LIN {X 0.099,Y -360.275,Z 1680.409,A 0.000,B 0.000,C 90.000,E1 73.630} C_DIS
LIN {X 0.182,Y -346.162,Z 1680.394,A 0.000,B 0.000,C 90.000,E1 70.913} C_DIS
LIN {X 0.106,Y -331.569,Z 1680.377,A 0.000,B 0.000,C 90.000,E1 67.847} C_DIS
LIN {X -0.099,Y -319.051,Z 1680.361,A 0.000,B 0.000,C 90.000,E1 65.049} C_DIS
LIN {X -0.146,Y -308.197,Z 1680.347,A 0.000,B 0.000,C 90.000,E1 62.487} C_DIS
LIN {X -0.186,Y -298.755,Z 1680.334,A 0.000,B 0.000,C 90.000,E1 60.205} C_DIS
LIN {X -0.133,Y -290.521,Z 1680.323,A 0.000,B 0.000,C 90.000,E1 58.201} C_DIS
LIN {X 0.074,Y -282.040,Z 1680.312,A 0.000,B 0.000,C 90.000,E1 56.135} C_DIS
LIN {X -0.110,Y -273.413,Z 1680.301,A 0.000,B 0.000,C 90.000,E1 54.116} C_DIS
LIN {X -0.060,Y -263.348,Z 1680.287,A 0.000,B 0.000,C 90.000,E1 51.662} C_DIS
LIN {X -0.034,Y -250.950,Z 1680.269,A 0.000,B 0.000,C 90.000,E1 48.447} C_DIS
LIN {X -0.049,Y -239.332,Z 1680.251,A 0.000,B 0.000,C 90.000,E1 45.162} C_DIS
LIN {X 0.006,Y -229.929,Z 1680.234,A 0.000,B 0.000,C 90.000,E1 42.162} C_DIS
LIN {X 0.085,Y -222.365,Z 1680.219,A 0.000,B 0.000,C 90.000,E1 39.483} C_DIS
LIN {X -0.012,Y -214.434,Z 1680.202,A 0.000,B 0.000,C 90.000,E1 36.423} C_DIS
LIN {X -0.034,Y -207.223,Z 1680.185,A 0.000,B 0.000,C 90.000,E1 33.293} C_DIS
LIN {X 0.067,Y -200.567,Z 1680.167,A 0.000,B 0.000,C 90.000,E1 30.079} C_DIS
LIN {X -0.020,Y -194.422,Z 1680.149,A 0.000,B 0.000,C 90.000,E1 26.873} C_DIS
LIN {X 0.005,Y -188.845,Z 1680.131,A 0.000,B 0.000,C 90.000,E1 23.590} C_DIS
LIN {X -0.084,Y -183.863,Z 1680.113,A 0.000,B 0.000,C 90.000,E1 20.301} C_DIS
LIN {X 0.028,Y -179.445,Z 1680.094,A 0.000,B 0.000,C 90.000,E1 16.913} C_DIS
LIN {X -0.003,Y -175.792,Z 1680.075,A 0.000,B 0.000,C 90.000,E1 13.536} C_DIS
LIN {X -0.006,Y -172.211,Z 1680.052,A 0.000,B 0.000,C 90.000,E1 9.265} C_DIS
LIN {X 0.053,Y -169.093,Z 1680.023,A 0.000,B 0.000,C 90.000,E1 4.073} C_DIS
LIN {X 0.081,Y -167.205,Z 1679.988,A 0.000,B 0.000,C 90.000,E1 357.764} C_DIS
LIN {X -0.016,Y -168.352,Z 1679.930,A 0.000,B 0.000,C 90.000,E1 347.353} C_DIS
LIN {X 0.061,Y -170.991,Z 1679.901,A 0.000,B 0.000,C 90.000,E1 342.127} C_DIS
LIN {X -0.022,Y -174.386,Z 1679.877,A 0.000,B 0.000,C 90.000,E1 337.847} C_DIS
LIN {X 0.038,Y -178.074,Z 1679.858,A 0.000,B 0.000,C 90.000,E1 334.409} C_DIS
LIN {X -0.065,Y -182.436,Z 1679.839,A 0.000,B 0.000,C 90.000,E1 331.051} C_DIS
LIN {X 0.050,Y -187.733,Z 1679.820,A 0.000,B 0.000,C 90.000,E1 327.661} C_DIS
LIN {X 0.015,Y -192.363,Z 1679.807,A 0.000,B 0.000,C 90.000,E1 325.182} C_DIS
LIN {X 0.016,Y -197.628,Z 1679.793,A 0.000,B 0.000,C 90.000,E1 322.718} C_DIS
LIN {X -0.080,Y -204.609,Z 1679.777,A 0.000,B 0.000,C 90.000,E1 319.908} C_DIS
LIN {X -0.032,Y -212.531,Z 1679.762,A 0.000,B 0.000,C 90.000,E1 317.106} C_DIS
LIN {X 0.028,Y -221.548,Z 1679.746,A 0.000,B 0.000,C 90.000,E1 314.352} C_DIS
LIN {X -0.018,Y -231.549,Z 1679.732,A 0.000,B 0.000,C 90.000,E1 311.676} C_DIS
LIN {X 0.050,Y -241.118,Z 1679.719,A 0.000,B 0.000,C 90.000,E1 309.402} C_DIS
LIN {X -0.006,Y -251.816,Z 1679.707,A 0.000,B 0.000,C 90.000,E1 307.202} C_DIS
LIN {X -0.009,Y -267.871,Z 1679.691,A 0.000,B 0.000,C 90.000,E1 304.326} C_DIS
LIN {X 0.014,Y -283.371,Z 1679.677,A 0.000,B 0.000,C 90.000,E1 301.878} C_DIS
LIN {X -0.162,Y -300.081,Z 1679.664,A 0.000,B 0.000,C 90.000,E1 299.539} C_DIS
LIN {X 0.012,Y -317.510,Z 1679.651,A 0.000,B 0.000,C 90.000,E1 297.206} C_DIS
LIN {X 0.091,Y -330.014,Z 1679.642,A 0.000,B 0.000,C 90.000,E1 295.591} C_DIS
LIN {X -0.088,Y -347.481,Z 1679.630,A 0.000,B 0.000,C 90.000,E1 293.439} C_DIS
LIN {X 0.040,Y -360.043,Z 1679.622,A 0.000,B 0.000,C 90.000,E1 291.897} C_DIS
LIN {X -0.092,Y -372.166,Z 1679.613,A 0.000,B 0.000,C 90.000,E1 290.429} C_DIS
LIN {X 0.075,Y -378.963,Z 1679.609,A 0.000,B 0.000,C 90.000,E1 289.523} C_DIS
LIN {X -0.042,Y -385.176,Z 1679.604,A 0.000,B 0.000,C 90.000,E1 288.671} C_DIS
LIN {X -0.115,Y -390.636,Z 1679.599,A 0.000,B 0.000,C 90.000,E1 287.819} C_DIS
LIN {X -0.137,Y -395.273,Z 1679.594,A 0.000,B 0.000,C 90.000,E1 286.968} C_DIS
LIN {X 0.145,Y -398.887,Z 1679.589,A 0.000,B 0.000,C 90.000,E1 286.079} C_DIS
LIN {X -0.099,Y -400.856,Z 1679.586,A 0.000,B 0.000,C 90.000,E1 285.552} C_DIS
LIN {X 0.157,Y -402.461,Z 1679.583,A 0.000,B 0.000,C 90.000,E1 284.954} C_DIS
LIN {X 0.034,Y -403.719,Z 1679.580,A 0.000,B 0.000,C 90.000,E1 284.411} C_DIS
LIN {X -0.182,Y -404.584,Z 1679.577,A 0.000,B 0.000,C 90.000,E1 283.883} C_DIS
LIN {X 0.006,Y -404.997,Z 1679.574,A 0.000,B 0.000,C 90.000,E1 283.300} C_DIS
LIN {X -0.195,Y -405.069,Z 1679.571,A 0.000,B 0.000,C 90.000,E1 282.771} C_DIS
LIN {X 0.004,Y -404.620,Z 1679.568,A 0.000,B 0.000,C 90.000,E1 282.187} C_DIS
LIN {X -0.192,Y -403.716,Z 1679.565,A 0.000,B 0.000,C 90.000,E1 281.658} C_DIS
LIN {X 0.004,Y -402.255,Z 1679.562,A 0.000,B 0.000,C 90.000,E1 281.074} C_DIS
LIN {X -0.200,Y -400.281,Z 1679.558,A 0.000,B 0.000,C 90.000,E1 280.546} C_DIS
LIN {X -0.021,Y -397.689,Z 1679.555,A 0.000,B 0.000,C 90.000,E1 279.962} C_DIS
LIN {X 0.135,Y -394.640,Z 1679.552,A 0.000,B 0.000,C 90.000,E1 279.378} C_DIS
LIN {X -0.119,Y -389.406,Z 1679.547,A 0.000,B 0.000,C 90.000,E1 278.568} C_DIS
LIN {X -0.025,Y -383.414,Z 1679.543,A 0.000,B 0.000,C 90.000,E1 277.701} C_DIS
LIN {X -0.008,Y -378.966,Z 1679.540,A 0.000,B 0.000,C 90.000,E1 277.125} C_DIS
LIN {X -0.016,Y -373.970,Z 1679.536,A 0.000,B 0.000,C 90.000,E1 276.549} C_DIS
LIN {X 0.069,Y -368.403,Z 1679.533,A 0.000,B 0.000,C 90.000,E1 275.967} C_DIS
LIN {X -0.036,Y -362.598,Z 1679.530,A 0.000,B 0.000,C 90.000,E1 275.454} C_DIS
LIN {X 0.114,Y -356.440,Z 1679.527,A 0.000,B 0.000,C 90.000,E1 274.935} C_DIS
LIN {X -0.154,Y -350.104,Z 1679.525,A 0.000,B 0.000,C 90.000,E1 274.531} C_DIS
LIN {X 0.146,Y -343.492,Z 1679.523,A 0.000,B 0.000,C 90.000,E1 274.073} C_DIS
LIN {X 0.093,Y -333.687,Z 1679.520,A 0.000,B 0.000,C 90.000,E1 273.555} C_DIS
LIN {X 0.060,Y -323.811,Z 1679.517,A 0.000,B 0.000,C 90.000,E1 273.094} C_DIS
LIN {X -0.012,Y -313.990,Z 1679.515,A 0.000,B 0.000,C 90.000,E1 272.694} C_DIS
LIN {X 0.146,Y -303.822,Z 1679.513,A 0.000,B 0.000,C 90.000,E1 272.293} C_DIS
LIN {X 0.009,Y -293.379,Z 1679.511,A 0.000,B 0.000,C 90.000,E1 272.007} C_DIS
LIN {X -0.132,Y -281.634,Z 1679.510,A 0.000,B 0.000,C 90.000,E1 271.776} C_DIS
LIN {X 0.036,Y -273.036,Z 1679.509,A 0.000,B 0.000,C 90.000,E1 271.604} C_DIS
LIN {X -0.021,Y -259.535,Z 1679.508,A 0.000,B 0.000,C 90.000,E1 271.489} C_DIS
LIN {X -0.031,Y -205.689,Z 1679.508,A 0.000,B 0.000,C 90.000,E1 271.375} C_DIS
LIN {X 0.019,Y -183.367,Z 1679.507,A 0.000,B 0.000,C 90.000,E1 271.260} C_DIS
LIN {X -0.015,Y -181.401,Z 1679.507,A 0.000,B 0.000,C 90.000,E1 271.260} C_DIS
LIN {X 0.026,Y -181.581,Z 1679.501,A 0.000,B 0.000,C 90.000,E1 270.229} C_DIS
LIN {X 0.030,Y -180.865,Z 1679.472,A 0.000,B 0.000,C 90.000,E1 265.008} C_DIS
LIN {X -0.094,Y -178.980,Z 1679.444,A 0.000,B 0.000,C 90.000,E1 259.982} C_DIS
LIN {X -0.082,Y -177.950,Z 1679.435,A 0.000,B 0.000,C 90.000,E1 258.285} C_DIS
LIN {X -0.062,Y -175.591,Z 1679.411,A 0.000,B 0.000,C 90.000,E1 254.031} C_DIS
LIN {X -0.050,Y -172.315,Z 1679.387,A 0.000,B 0.000,C 90.000,E1 249.752} C_DIS
LIN {X -0.071,Y -171.794,Z 1679.383,A 0.000,B 0.000,C 90.000,E1 248.901} C_DIS
LIN {X -0.033,Y -169.464,Z 1679.368,A 0.000,B 0.000,C 90.000,E1 246.305} C_DIS
LIN {X 0.023,Y -166.792,Z 1679.349,A 0.000,B 0.000,C 90.000,E1 242.820} C_DIS
LIN {X 0.018,Y -162.773,Z 1679.325,A 0.000,B 0.000,C 90.000,E1 238.456} C_DIS
LIN {X -0.006,Y -161.462,Z 1679.315,A 0.000,B 0.000,C 90.000,E1 236.707} C_DIS
LIN {X 0.035,Y -157.456,Z 1679.290,A 0.000,B 0.000,C 90.000,E1 232.271} C_DIS
LIN {X -0.032,Y -155.468,Z 1679.276,A 0.000,B 0.000,C 90.000,E1 229.622} C_DIS
LIN {X 0.009,Y -151.781,Z 1679.251,A 0.000,B 0.000,C 90.000,E1 225.121} C_DIS
LIN {X 0.026,Y -149.986,Z 1679.236,A 0.000,B 0.000,C 90.000,E1 222.405} C_DIS
LIN {X -0.053,Y -146.819,Z 1679.210,A 0.000,B 0.000,C 90.000,E1 217.890} C_DIS
LIN {X 0.053,Y -145.398,Z 1679.195,A 0.000,B 0.000,C 90.000,E1 215.105} C_DIS
LIN {X -0.030,Y -142.832,Z 1679.170,A 0.000,B 0.000,C 90.000,E1 210.541} C_DIS
LIN {X 0.026,Y -141.445,Z 1679.149,A 0.000,B 0.000,C 90.000,E1 206.821} C_DIS
LIN {X 0.071,Y -139.369,Z 1679.113,A 0.000,B 0.000,C 90.000,E1 200.301} C_DIS
LIN {X 0.058,Y -138.817,Z 1679.097,A 0.000,B 0.000,C 90.000,E1 197.511} C_DIS
LIN {X -0.028,Y -138.352,Z 1679.056,A 0.000,B 0.000,C 90.000,E1 190.074} C_DIS
LIN {X -0.055,Y -139.536,Z 1679.004,A 0.000,B 0.000,C 90.000,E1 180.745} C_DIS
LIN {X 0.038,Y -141.223,Z 1678.973,A 0.000,B 0.000,C 90.000,E1 175.122} C_DIS
LIN {X -0.004,Y -142.596,Z 1678.958,A 0.000,B 0.000,C 90.000,E1 172.356} C_DIS
LIN {X -0.050,Y -144.900,Z 1678.932,A 0.000,B 0.000,C 90.000,E1 167.757} C_DIS
LIN {X 0.044,Y -147.528,Z 1678.911,A 0.000,B 0.000,C 90.000,E1 164.047} C_DIS
LIN {X -0.023,Y -150.125,Z 1678.891,A 0.000,B 0.000,C 90.000,E1 160.423} C_DIS
LIN {X -0.013,Y -153.488,Z 1678.871,A 0.000,B 0.000,C 90.000,E1 156.794} C_DIS
LIN {X 0.051,Y -157.852,Z 1678.846,A 0.000,B 0.000,C 90.000,E1 152.281} C_DIS
LIN {X 0.007,Y -162.138,Z 1678.826,A 0.000,B 0.000,C 90.000,E1 148.742} C_DIS
LIN {X -0.014,Y -166.341,Z 1678.807,A 0.000,B 0.000,C 90.000,E1 145.229} C_DIS
LIN {X -0.008,Y -171.359,Z 1678.787,A 0.000,B 0.000,C 90.000,E1 141.743} C_DIS
LIN {X -0.081,Y -176.265,Z 1678.768,A 0.000,B 0.000,C 90.000,E1 138.324} C_DIS
LIN {X 0.038,Y -180.548,Z 1678.754,A 0.000,B 0.000,C 90.000,E1 135.729} C_DIS
LIN {X 0.017,Y -185.950,Z 1678.735,A 0.000,B 0.000,C 90.000,E1 132.366} C_DIS
LIN {X -0.049,Y -190.581,Z 1678.722,A 0.000,B 0.000,C 90.000,E1 129.886} C_DIS
LIN {X -0.019,Y -196.331,Z 1678.703,A 0.000,B 0.000,C 90.000,E1 126.583} C_DIS
LIN {X 0.058,Y -201.128,Z 1678.690,A 0.000,B 0.000,C 90.000,E1 124.119} C_DIS
LIN {X 0.071,Y -207.431,Z 1678.671,A 0.000,B 0.000,C 90.000,E1 120.718} C_DIS
LIN {X 0.032,Y -208.076,Z 1678.669,A 0.000,B 0.000,C 90.000,E1 120.413} C_DIS
LIN {X 0.003,Y -329.906,Z 1678.669,A 0.000,B 0.000,C 90.000,E1 120.413} C_DIS
LIN {X 0.063,Y -335.128,Z 1678.668,A 0.000,B 0.000,C 90.000,E1 120.256} C_DIS
LIN {X -0.047,Y -337.460,Z 1678.667,A 0.000,B 0.000,C 90.000,E1 120.129} C_DIS
LIN {X -0.010,Y -341.319,Z 1678.665,A 0.000,B 0.000,C 90.000,E1 119.745} C_DIS
LIN {X -0.018,Y -344.755,Z 1678.662,A 0.000,B 0.000,C 90.000,E1 119.205} C_DIS
LIN {X 0.025,Y -358.759,Z 1678.645,A 0.000,B 0.000,C 90.000,E1 116.155} C_DIS
LIN {X 0.143,Y -372.868,Z 1678.630,A 0.000,B 0.000,C 90.000,E1 113.462} C_DIS
LIN {X 0.031,Y -386.769,Z 1678.618,A 0.000,B 0.000,C 90.000,E1 111.153} C_DIS
LIN {X -0.168,Y -402.046,Z 1678.605,A 0.000,B 0.000,C 90.000,E1 108.906} C_DIS
LIN {X -0.121,Y -418.806,Z 1678.593,A 0.000,B 0.000,C 90.000,E1 106.677} C_DIS
LIN {X 0.111,Y -437.163,Z 1678.581,A 0.000,B 0.000,C 90.000,E1 104.481} C_DIS
LIN {X 0.096,Y -456.905,Z 1678.569,A 0.000,B 0.000,C 90.000,E1 102.411} C_DIS
LIN {X 0.210,Y -477.250,Z 1678.558,A 0.000,B 0.000,C 90.000,E1 100.489} C_DIS
LIN {X 0.010,Y -503.191,Z 1678.546,A 0.000,B 0.000,C 90.000,E1 98.341} C_DIS
LIN {X -0.236,Y -505.054,Z 1678.545,A 0.000,B 0.000,C 90.000,E1 98.163} C_DIS
LIN {X 0.201,Y -506.717,Z 1678.544,A 0.000,B 0.000,C 90.000,E1 97.871} C_DIS
LIN {X 0.068,Y -507.959,Z 1678.542,A 0.000,B 0.000,C 90.000,E1 97.644} C_DIS
LIN {X -0.109,Y -509.463,Z 1678.540,A 0.000,B 0.000,C 90.000,E1 97.182} C_DIS
LIN {X 0.228,Y -509.885,Z 1678.537,A 0.000,B 0.000,C 90.000,E1 96.663} C_DIS
LIN {X 0.066,Y -509.297,Z 1678.535,A 0.000,B 0.000,C 90.000,E1 96.201} C_DIS
LIN {X -0.095,Y -507.598,Z 1678.532,A 0.000,B 0.000,C 90.000,E1 95.739} C_DIS
LIN {X -0.201,Y -506.231,Z 1678.531,A 0.000,B 0.000,C 90.000,E1 95.511} C_DIS
LIN {X 0.226,Y -495.749,Z 1678.522,A 0.000,B 0.000,C 90.000,E1 94.012} C_DIS
LIN {X 0.238,Y -483.294,Z 1678.513,A 0.000,B 0.000,C 90.000,E1 92.293} C_DIS
LIN {X 0.194,Y -472.512,Z 1678.505,A 0.000,B 0.000,C 90.000,E1 90.802} C_DIS
LIN {X 0.213,Y -459.844,Z 1678.495,A 0.000,B 0.000,C 90.000,E1 89.026} C_DIS
LIN {X -0.214,Y -448.803,Z 1678.486,A 0.000,B 0.000,C 90.000,E1 87.535} C_DIS
LIN {X 0.094,Y -437.446,Z 1678.477,A 0.000,B 0.000,C 90.000,E1 85.927} C_DIS
LIN {X -0.104,Y -424.099,Z 1678.467,A 0.000,B 0.000,C 90.000,E1 84.090} C_DIS
LIN {X 0.164,Y -407.287,Z 1678.453,A 0.000,B 0.000,C 90.000,E1 81.602} C_DIS
LIN {X 0.176,Y -387.882,Z 1678.436,A 0.000,B 0.000,C 90.000,E1 78.522} C_DIS
LIN {X 0.155,Y -372.717,Z 1678.422,A 0.000,B 0.000,C 90.000,E1 75.936} C_DIS
LIN {X -0.037,Y -359.758,Z 1678.409,A 0.000,B 0.000,C 90.000,E1 73.614} C_DIS
LIN {X -0.061,Y -345.645,Z 1678.394,A 0.000,B 0.000,C 90.000,E1 70.913} C_DIS
LIN {X -0.128,Y -332.511,Z 1678.379,A 0.000,B 0.000,C 90.000,E1 68.156} C_DIS
LIN {X -0.001,Y -319.952,Z 1678.363,A 0.000,B 0.000,C 90.000,E1 65.305} C_DIS
LIN {X -0.031,Y -309.082,Z 1678.349,A 0.000,B 0.000,C 90.000,E1 62.743} C_DIS
LIN {X -0.081,Y -301.015,Z 1678.338,A 0.000,B 0.000,C 90.000,E1 60.795} C_DIS
LIN {X 0.014,Y -292.798,Z 1678.327,A 0.000,B 0.000,C 90.000,E1 58.791} C_DIS
LIN {X -0.048,Y -284.359,Z 1678.315,A 0.000,B 0.000,C 90.000,E1 56.786} C_DIS
LIN {X -0.034,Y -275.737,Z 1678.304,A 0.000,B 0.000,C 90.000,E1 54.736} C_DIS
LIN {X 0.117,Y -265.658,Z 1678.291,A 0.000,B 0.000,C 90.000,E1 52.271} C_DIS
LIN {X 0.025,Y -253.124,Z 1678.273,A 0.000,B 0.000,C 90.000,E1 49.094} C_DIS
LIN {X 0.062,Y -241.385,Z 1678.255,A 0.000,B 0.000,C 90.000,E1 45.810} C_DIS
LIN {X -0.007,Y -231.825,Z 1678.238,A 0.000,B 0.000,C 90.000,E1 42.852} C_DIS
LIN {X 0.000,Y -222.065,Z 1678.219,A 0.000,B 0.000,C 90.000,E1 39.439} C_DIS
LIN {X -0.094,Y -214.179,Z 1678.202,A 0.000,B 0.000,C 90.000,E1 36.377} C_DIS
LIN {X 0.001,Y -206.993,Z 1678.185,A 0.000,B 0.000,C 90.000,E1 33.214} C_DIS
LIN {X 0.092,Y -200.341,Z 1678.167,A 0.000,B 0.000,C 90.000,E1 30.001} C_DIS
LIN {X -0.006,Y -194.206,Z 1678.149,A 0.000,B 0.000,C 90.000,E1 26.796} C_DIS
LIN {X 0.007,Y -188.633,Z 1678.131,A 0.000,B 0.000,C 90.000,E1 23.515} C_DIS
LIN {X 0.017,Y -183.668,Z 1678.112,A 0.000,B 0.000,C 90.000,E1 20.194} C_DIS
LIN {X -0.044,Y -179.265,Z 1678.094,A 0.000,B 0.000,C 90.000,E1 16.858} C_DIS
LIN {X -0.033,Y -175.630,Z 1678.075,A 0.000,B 0.000,C 90.000,E1 13.467} C_DIS
LIN {X -0.078,Y -172.093,Z 1678.051,A 0.000,B 0.000,C 90.000,E1 9.208} C_DIS
LIN {X -0.008,Y -169.022,Z 1678.022,A 0.000,B 0.000,C 90.000,E1 4.012} C_DIS
LIN {X 0.046,Y -167.088,Z 1677.983,A 0.000,B 0.000,C 90.000,E1 356.906} C_DIS
LIN {X -0.017,Y -168.346,Z 1677.930,A 0.000,B 0.000,C 90.000,E1 347.353} C_DIS
LIN {X 0.060,Y -171.007,Z 1677.901,A 0.000,B 0.000,C 90.000,E1 342.127} C_DIS
LIN {X -0.023,Y -174.421,Z 1677.877,A 0.000,B 0.000,C 90.000,E1 337.847} C_DIS
LIN {X 0.037,Y -178.135,Z 1677.858,A 0.000,B 0.000,C 90.000,E1 334.409} C_DIS
LIN {X -0.062,Y -182.525,Z 1677.839,A 0.000,B 0.000,C 90.000,E1 331.051} C_DIS
LIN {X 0.054,Y -187.855,Z 1677.820,A 0.000,B 0.000,C 90.000,E1 327.661} C_DIS
LIN {X 0.023,Y -192.490,Z 1677.807,A 0.000,B 0.000,C 90.000,E1 325.182} C_DIS
LIN {X 0.026,Y -197.778,Z 1677.793,A 0.000,B 0.000,C 90.000,E1 322.718} C_DIS
LIN {X -0.061,Y -204.778,Z 1677.777,A 0.000,B 0.000,C 90.000,E1 319.908} C_DIS
LIN {X -0.008,Y -212.704,Z 1677.762,A 0.000,B 0.000,C 90.000,E1 317.106} C_DIS
LIN {X 0.056,Y -221.721,Z 1677.746,A 0.000,B 0.000,C 90.000,E1 314.352} C_DIS
LIN {X 0.016,Y -231.721,Z 1677.732,A 0.000,B 0.000,C 90.000,E1 311.676} C_DIS
LIN {X 0.069,Y -242.978,Z 1677.717,A 0.000,B 0.000,C 90.000,E1 309.036} C_DIS
LIN {X -0.115,Y -251.980,Z 1677.707,A 0.000,B 0.000,C 90.000,E1 307.237} C_DIS
LIN {X -0.008,Y -265.884,Z 1677.693,A 0.000,B 0.000,C 90.000,E1 304.692} C_DIS
LIN {X 0.118,Y -281.162,Z 1677.679,A 0.000,B 0.000,C 90.000,E1 302.212} C_DIS
LIN {X -0.093,Y -297.733,Z 1677.666,A 0.000,B 0.000,C 90.000,E1 299.873} C_DIS
LIN {X 0.168,Y -315.047,Z 1677.653,A 0.000,B 0.000,C 90.000,E1 297.513} C_DIS
LIN {X 0.076,Y -327.594,Z 1677.644,A 0.000,B 0.000,C 90.000,E1 295.924} C_DIS
LIN {X -0.146,Y -342.500,Z 1677.634,A 0.000,B 0.000,C 90.000,E1 294.079} C_DIS
LIN {X 0.078,Y -357.549,Z 1677.623,A 0.000,B 0.000,C 90.000,E1 292.206} C_DIS
LIN {X -0.099,Y -369.784,Z 1677.615,A 0.000,B 0.000,C 90.000,E1 290.737} C_DIS
LIN {X 0.179,Y -376.720,Z 1677.610,A 0.000,B 0.000,C 90.000,E1 289.812} C_DIS
LIN {X 0.032,Y -383.129,Z 1677.605,A 0.000,B 0.000,C 90.000,E1 288.960} C_DIS
LIN {X -0.054,Y -388.887,Z 1677.601,A 0.000,B 0.000,C 90.000,E1 288.109} C_DIS
LIN {X 0.123,Y -392.279,Z 1677.597,A 0.000,B 0.000,C 90.000,E1 287.511} C_DIS
LIN {X -0.003,Y -396.578,Z 1677.593,A 0.000,B 0.000,C 90.000,E1 286.677} C_DIS
LIN {X -0.153,Y -398.928,Z 1677.589,A 0.000,B 0.000,C 90.000,E1 286.134} C_DIS
LIN {X -0.014,Y -400.922,Z 1677.586,A 0.000,B 0.000,C 90.000,E1 285.552} C_DIS
LIN {X -0.145,Y -402.560,Z 1677.583,A 0.000,B 0.000,C 90.000,E1 285.009} C_DIS
LIN {X 0.021,Y -403.847,Z 1677.580,A 0.000,B 0.000,C 90.000,E1 284.426} C_DIS
LIN {X -0.094,Y -404.703,Z 1677.577,A 0.000,B 0.000,C 90.000,E1 283.883} C_DIS
LIN {X 0.094,Y -405.165,Z 1677.574,A 0.000,B 0.000,C 90.000,E1 283.300} C_DIS
LIN {X -0.105,Y -405.194,Z 1677.571,A 0.000,B 0.000,C 90.000,E1 282.771} C_DIS
LIN {X 0.094,Y -404.813,Z 1677.568,A 0.000,B 0.000,C 90.000,E1 282.187} C_DIS
LIN {X -0.101,Y -403.913,Z 1677.565,A 0.000,B 0.000,C 90.000,E1 281.658} C_DIS
LIN {X 0.096,Y -402.483,Z 1677.562,A 0.000,B 0.000,C 90.000,E1 281.074} C_DIS
LIN {X -0.107,Y -400.526,Z 1677.558,A 0.000,B 0.000,C 90.000,E1 280.546} C_DIS
LIN {X 0.072,Y -397.995,Z 1677.555,A 0.000,B 0.000,C 90.000,E1 279.962} C_DIS
LIN {X -0.154,Y -393.193,Z 1677.551,A 0.000,B 0.000,C 90.000,E1 279.151} C_DIS
LIN {X 0.033,Y -387.680,Z 1677.546,A 0.000,B 0.000,C 90.000,E1 278.276} C_DIS
LIN {X 0.103,Y -381.468,Z 1677.541,A 0.000,B 0.000,C 90.000,E1 277.409} C_DIS
LIN {X 0.105,Y -376.753,Z 1677.538,A 0.000,B 0.000,C 90.000,E1 276.834} C_DIS
LIN {X 0.117,Y -371.379,Z 1677.535,A 0.000,B 0.000,C 90.000,E1 276.258} C_DIS
LIN {X -0.096,Y -365.609,Z 1677.532,A 0.000,B 0.000,C 90.000,E1 275.739} C_DIS
LIN {X -0.060,Y -359.612,Z 1677.529,A 0.000,B 0.000,C 90.000,E1 275.220} C_DIS
LIN {X -0.086,Y -353.351,Z 1677.526,A 0.000,B 0.000,C 90.000,E1 274.759} C_DIS
LIN {X 0.132,Y -346.946,Z 1677.524,A 0.000,B 0.000,C 90.000,E1 274.302} C_DIS
LIN {X -0.075,Y -337.053,Z 1677.521,A 0.000,B 0.000,C 90.000,E1 273.784} C_DIS
LIN {X 0.154,Y -327.473,Z 1677.518,A 0.000,B 0.000,C 90.000,E1 273.269} C_DIS
LIN {X -0.013,Y -317.642,Z 1677.516,A 0.000,B 0.000,C 90.000,E1 272.865} C_DIS
LIN {X 0.082,Y -307.798,Z 1677.514,A 0.000,B 0.000,C 90.000,E1 272.465} C_DIS
LIN {X 0.084,Y -297.334,Z 1677.512,A 0.000,B 0.000,C 90.000,E1 272.121} C_DIS
LIN {X -0.018,Y -290.098,Z 1677.511,A 0.000,B 0.000,C 90.000,E1 271.949} C_DIS
LIN {X -0.042,Y -278.053,Z 1677.510,A 0.000,B 0.000,C 90.000,E1 271.718} C_DIS
LIN {X 0.038,Y -265.606,Z 1677.509,A 0.000,B 0.000,C 90.000,E1 271.547} C_DIS
LIN {X 0.021,Y -249.623,Z 1677.508,A 0.000,B 0.000,C 90.000,E1 271.489} C_DIS
LIN {X -0.114,Y -237.343,Z 1677.508,A 0.000,B 0.000,C 90.000,E1 271.489} C_DIS
LIN {X 0.076,Y -230.146,Z 1677.508,A 0.000,B 0.000,C 90.000,E1 271.432} C_DIS
LIN {X 0.054,Y -194.600,Z 1677.507,A 0.000,B 0.000,C 90.000,E1 271.318} C_DIS
LIN {X 0.054,Y -183.332,Z 1677.507,A 0.000,B 0.000,C 90.000,E1 271.260} C_DIS
LIN {X 0.017,Y -181.398,Z 1677.507,A 0.000,B 0.000,C 90.000,E1 271.260} C_DIS
LIN {X 0.000,Y -181.575,Z 1677.502,A 0.000,B 0.000,C 90.000,E1 270.401} C_DIS
LIN {X -0.023,Y -180.906,Z 1677.474,A 0.000,B 0.000,C 90.000,E1 265.355} C_DIS
LIN {X 0.051,Y -180.678,Z 1677.469,A 0.000,B 0.000,C 90.000,E1 264.489} C_DIS
LIN {X -0.051,Y -178.761,Z 1677.441,A 0.000,B 0.000,C 90.000,E1 259.454} C_DIS
LIN {X 0.022,Y -175.808,Z 1677.413,A 0.000,B 0.000,C 90.000,E1 254.338} C_DIS
LIN {X 0.016,Y -171.993,Z 1677.385,A 0.000,B 0.000,C 90.000,E1 249.209} C_DIS
LIN {X 0.054,Y -171.404,Z 1677.380,A 0.000,B 0.000,C 90.000,E1 248.337} C_DIS
LIN {X 0.038,Y -167.646,Z 1677.356,A 0.000,B 0.000,C 90.000,E1 244.024} C_DIS
LIN {X 0.054,Y -166.308,Z 1677.346,A 0.000,B 0.000,C 90.000,E1 242.281} C_DIS
LIN {X 0.047,Y -163.051,Z 1677.327,A 0.000,B 0.000,C 90.000,E1 238.791} C_DIS
LIN {X 0.008,Y -160.985,Z 1677.312,A 0.000,B 0.000,C 90.000,E1 236.167} C_DIS
LIN {X -0.014,Y -157.734,Z 1677.292,A 0.000,B 0.000,C 90.000,E1 232.637} C_DIS
LIN {X -0.076,Y -155.773,Z 1677.278,A 0.000,B 0.000,C 90.000,E1 229.989} C_DIS
LIN {X -0.020,Y -152.028,Z 1677.253,A 0.000,B 0.000,C 90.000,E1 225.486} C_DIS
LIN {X -0.002,Y -150.276,Z 1677.238,A 0.000,B 0.000,C 90.000,E1 222.771} C_DIS
LIN {X 0.015,Y -147.026,Z 1677.212,A 0.000,B 0.000,C 90.000,E1 218.222} C_DIS
LIN {X 0.035,Y -145.608,Z 1677.197,A 0.000,B 0.000,C 90.000,E1 215.471} C_DIS
LIN {X 0.040,Y -142.993,Z 1677.172,A 0.000,B 0.000,C 90.000,E1 210.875} C_DIS
LIN {X -0.025,Y -141.621,Z 1677.151,A 0.000,B 0.000,C 90.000,E1 207.206} C_DIS
LIN {X 0.031,Y -139.431,Z 1677.115,A 0.000,B 0.000,C 90.000,E1 200.684} C_DIS
LIN {X -0.046,Y -139.161,Z 1677.105,A 0.000,B 0.000,C 90.000,E1 198.852} C_DIS
LIN {X -0.009,Y -138.341,Z 1677.058,A 0.000,B 0.000,C 90.000,E1 190.433} C_DIS
LIN {X -0.001,Y -139.479,Z 1677.006,A 0.000,B 0.000,C 90.000,E1 181.088} C_DIS
LIN {X -0.061,Y -141.065,Z 1676.975,A 0.000,B 0.000,C 90.000,E1 175.527} C_DIS
LIN {X 0.034,Y -142.440,Z 1676.960,A 0.000,B 0.000,C 90.000,E1 172.704} C_DIS
LIN {X -0.046,Y -144.678,Z 1676.934,A 0.000,B 0.000,C 90.000,E1 168.117} C_DIS
LIN {X 0.078,Y -147.268,Z 1676.913,A 0.000,B 0.000,C 90.000,E1 164.393} C_DIS
LIN {X -0.046,Y -150.585,Z 1676.888,A 0.000,B 0.000,C 90.000,E1 159.880} C_DIS
LIN {X 0.032,Y -154.056,Z 1676.868,A 0.000,B 0.000,C 90.000,E1 156.230} C_DIS
LIN {X -0.042,Y -157.475,Z 1676.848,A 0.000,B 0.000,C 90.000,E1 152.666} C_DIS
LIN {X 0.045,Y -161.698,Z 1676.828,A 0.000,B 0.000,C 90.000,E1 149.076} C_DIS
LIN {X -0.077,Y -165.893,Z 1676.809,A 0.000,B 0.000,C 90.000,E1 145.595} C_DIS
LIN {X 0.048,Y -170.874,Z 1676.789,A 0.000,B 0.000,C 90.000,E1 142.065} C_DIS
LIN {X 0.075,Y -175.743,Z 1676.770,A 0.000,B 0.000,C 90.000,E1 138.609} C_DIS
LIN {X -0.052,Y -181.354,Z 1676.751,A 0.000,B 0.000,C 90.000,E1 135.243} C_DIS
LIN {X 0.082,Y -186.844,Z 1676.733,A 0.000,B 0.000,C 90.000,E1 131.838} C_DIS
LIN {X 0.035,Y -191.431,Z 1676.719,A 0.000,B 0.000,C 90.000,E1 129.358} C_DIS
LIN {X -0.032,Y -197.282,Z 1676.700,A 0.000,B 0.000,C 90.000,E1 126.091} C_DIS
LIN {X 0.005,Y -200.560,Z 1676.691,A 0.000,B 0.000,C 90.000,E1 124.452} C_DIS
LIN {X -0.051,Y -207.599,Z 1676.670,A 0.000,B 0.000,C 90.000,E1 120.669} C_DIS
LIN {X -0.017,Y -208.003,Z 1676.669,A 0.000,B 0.000,C 90.000,E1 120.463} C_DIS
LIN {X -0.062,Y -329.589,Z 1676.669,A 0.000,B 0.000,C 90.000,E1 120.463} C_DIS
LIN {X -0.168,Y -331.226,Z 1676.669,A 0.000,B 0.000,C 90.000,E1 120.463} C_DIS
LIN {X -0.050,Y -334.512,Z 1676.668,A 0.000,B 0.000,C 90.000,E1 120.335} C_DIS
LIN {X -0.044,Y -337.760,Z 1676.667,A 0.000,B 0.000,C 90.000,E1 120.129} C_DIS
LIN {X -0.016,Y -341.442,Z 1676.665,A 0.000,B 0.000,C 90.000,E1 119.745} C_DIS
LIN {X 0.002,Y -343.357,Z 1676.664,A 0.000,B 0.000,C 90.000,E1 119.461} C_DIS
LIN {X -0.149,Y -344.862,Z 1676.662,A 0.000,B 0.000,C 90.000,E1 119.205} C_DIS
LIN {X -0.097,Y -358.832,Z 1676.645,A 0.000,B 0.000,C 90.000,E1 116.155} C_DIS
LIN {X 0.018,Y -372.951,Z 1676.630,A 0.000,B 0.000,C 90.000,E1 113.462} C_DIS
LIN {X -0.096,Y -386.863,Z 1676.617,A 0.000,B 0.000,C 90.000,E1 111.153} C_DIS
LIN {X 0.083,Y -402.152,Z 1676.605,A 0.000,B 0.000,C 90.000,E1 108.852} C_DIS
LIN {X 0.149,Y -418.924,Z 1676.592,A 0.000,B 0.000,C 90.000,E1 106.622} C_DIS
LIN {X -0.023,Y -437.295,Z 1676.580,A 0.000,B 0.000,C 90.000,E1 104.481} C_DIS
LIN {X -0.035,Y -457.042,Z 1676.569,A 0.000,B 0.000,C 90.000,E1 102.411} C_DIS
LIN {X 0.083,Y -477.392,Z 1676.558,A 0.000,B 0.000,C 90.000,E1 100.489} C_DIS
LIN {X 0.205,Y -500.894,Z 1676.547,A 0.000,B 0.000,C 90.000,E1 98.511} C_DIS
LIN {X -0.112,Y -503.264,Z 1676.546,A 0.000,B 0.000,C 90.000,E1 98.341} C_DIS
LIN {X 0.142,Y -505.060,Z 1676.545,A 0.000,B 0.000,C 90.000,E1 98.106} C_DIS
LIN {X 0.080,Y -506.666,Z 1676.544,A 0.000,B 0.000,C 90.000,E1 97.871} C_DIS
LIN {X -0.053,Y -507.864,Z 1676.542,A 0.000,B 0.000,C 90.000,E1 97.644} C_DIS
LIN {X -0.230,Y -509.300,Z 1676.540,A 0.000,B 0.000,C 90.000,E1 97.182} C_DIS
LIN {X 0.105,Y -509.665,Z 1676.537,A 0.000,B 0.000,C 90.000,E1 96.663} C_DIS
LIN {X -0.058,Y -509.018,Z 1676.534,A 0.000,B 0.000,C 90.000,E1 96.201} C_DIS
LIN {X -0.218,Y -507.247,Z 1676.532,A 0.000,B 0.000,C 90.000,E1 95.739} C_DIS
LIN {X 0.179,Y -505.833,Z 1676.530,A 0.000,B 0.000,C 90.000,E1 95.454} C_DIS
LIN {X -0.032,Y -493.596,Z 1676.521,A 0.000,B 0.000,C 90.000,E1 93.784} C_DIS
LIN {X -0.056,Y -481.130,Z 1676.511,A 0.000,B 0.000,C 90.000,E1 92.064} C_DIS
LIN {X -0.127,Y -470.321,Z 1676.503,A 0.000,B 0.000,C 90.000,E1 90.573} C_DIS
LIN {X -0.138,Y -457.664,Z 1676.493,A 0.000,B 0.000,C 90.000,E1 88.797} C_DIS
LIN {X -0.147,Y -446.567,Z 1676.485,A 0.000,B 0.000,C 90.000,E1 87.249} C_DIS
LIN {X 0.116,Y -435.128,Z 1676.476,A 0.000,B 0.000,C 90.000,E1 85.641} C_DIS
LIN {X -0.096,Y -421.778,Z 1676.465,A 0.000,B 0.000,C 90.000,E1 83.799} C_DIS
LIN {X 0.063,Y -405.027,Z 1676.452,A 0.000,B 0.000,C 90.000,E1 81.319} C_DIS
LIN {X 0.063,Y -385.738,Z 1676.435,A 0.000,B 0.000,C 90.000,E1 78.229} C_DIS
LIN {X -0.007,Y -370.629,Z 1676.420,A 0.000,B 0.000,C 90.000,E1 75.644} C_DIS
LIN {X 0.148,Y -356.115,Z 1676.406,A 0.000,B 0.000,C 90.000,E1 72.960} C_DIS
LIN {X 0.028,Y -339.280,Z 1676.387,A 0.000,B 0.000,C 90.000,E1 69.645} C_DIS
LIN {X -0.065,Y -327.812,Z 1676.373,A 0.000,B 0.000,C 90.000,E1 67.177} C_DIS
LIN {X -0.171,Y -316.805,Z 1676.359,A 0.000,B 0.000,C 90.000,E1 64.665} C_DIS
LIN {X 0.145,Y -306.006,Z 1676.345,A 0.000,B 0.000,C 90.000,E1 62.025} C_DIS
LIN {X 0.033,Y -297.887,Z 1676.334,A 0.000,B 0.000,C 90.000,E1 60.078} C_DIS
LIN {X 0.062,Y -289.591,Z 1676.323,A 0.000,B 0.000,C 90.000,E1 58.074} C_DIS
LIN {X -0.148,Y -281.045,Z 1676.311,A 0.000,B 0.000,C 90.000,E1 56.087} C_DIS
LIN {X 0.123,Y -270.915,Z 1676.298,A 0.000,B 0.000,C 90.000,E1 53.623} C_DIS
LIN {X -0.035,Y -259.526,Z 1676.282,A 0.000,B 0.000,C 90.000,E1 50.848} C_DIS
LIN {X -0.119,Y -247.383,Z 1676.265,A 0.000,B 0.000,C 90.000,E1 47.634} C_DIS
LIN {X 0.097,Y -236.133,Z 1676.246,A 0.000,B 0.000,C 90.000,E1 44.271} C_DIS
LIN {X 0.013,Y -225.992,Z 1676.227,A 0.000,B 0.000,C 90.000,E1 40.906} C_DIS
LIN {X -0.028,Y -217.810,Z 1676.210,A 0.000,B 0.000,C 90.000,E1 37.855} C_DIS
LIN {X -0.021,Y -210.297,Z 1676.193,A 0.000,B 0.000,C 90.000,E1 34.739} C_DIS
LIN {X -0.085,Y -203.395,Z 1676.175,A 0.000,B 0.000,C 90.000,E1 31.592} C_DIS
LIN {X -0.007,Y -196.977,Z 1676.158,A 0.000,B 0.000,C 90.000,E1 28.359} C_DIS
LIN {X 0.069,Y -191.146,Z 1676.139,A 0.000,B 0.000,C 90.000,E1 25.079} C_DIS
LIN {X 0.032,Y -185.892,Z 1676.121,A 0.000,B 0.000,C 90.000,E1 21.791} C_DIS
LIN {X -0.028,Y -181.198,Z 1676.103,A 0.000,B 0.000,C 90.000,E1 18.471} C_DIS
LIN {X 0.076,Y -177.204,Z 1676.084,A 0.000,B 0.000,C 90.000,E1 15.064} C_DIS
LIN {X -0.025,Y -173.260,Z 1676.060,A 0.000,B 0.000,C 90.000,E1 10.838} C_DIS
LIN {X -0.034,Y -169.857,Z 1676.031,A 0.000,B 0.000,C 90.000,E1 5.682} C_DIS
LIN {X -0.030,Y -167.459,Z 1675.997,A 0.000,B 0.000,C 90.000,E1 359.542} C_DIS
LIN {X -0.018,Y -168.335,Z 1675.930,A 0.000,B 0.000,C 90.000,E1 347.353} C_DIS
LIN {X 0.058,Y -171.020,Z 1675.901,A 0.000,B 0.000,C 90.000,E1 342.127} C_DIS
LIN {X -0.023,Y -174.458,Z 1675.877,A 0.000,B 0.000,C 90.000,E1 337.847} C_DIS
LIN {X 0.039,Y -178.198,Z 1675.858,A 0.000,B 0.000,C 90.000,E1 334.409} C_DIS
LIN {X -0.061,Y -182.630,Z 1675.839,A 0.000,B 0.000,C 90.000,E1 331.051} C_DIS
LIN {X 0.060,Y -187.982,Z 1675.820,A 0.000,B 0.000,C 90.000,E1 327.661} C_DIS
LIN {X 0.030,Y -192.625,Z 1675.807,A 0.000,B 0.000,C 90.000,E1 325.182} C_DIS
LIN {X 0.035,Y -197.923,Z 1675.793,A 0.000,B 0.000,C 90.000,E1 322.718} C_DIS
LIN {X -0.047,Y -204.954,Z 1675.777,A 0.000,B 0.000,C 90.000,E1 319.908} C_DIS
LIN {X 0.011,Y -212.882,Z 1675.762,A 0.000,B 0.000,C 90.000,E1 317.106} C_DIS
LIN {X 0.080,Y -221.894,Z 1675.746,A 0.000,B 0.000,C 90.000,E1 314.352} C_DIS
LIN {X 0.044,Y -231.907,Z 1675.732,A 0.000,B 0.000,C 90.000,E1 311.676} C_DIS
LIN {X -0.049,Y -243.129,Z 1675.717,A 0.000,B 0.000,C 90.000,E1 309.072} C_DIS
LIN {X -0.077,Y -252.132,Z 1675.707,A 0.000,B 0.000,C 90.000,E1 307.237} C_DIS
LIN {X 0.086,Y -268.111,Z 1675.691,A 0.000,B 0.000,C 90.000,E1 304.326} C_DIS
LIN {X -0.071,Y -281.262,Z 1675.679,A 0.000,B 0.000,C 90.000,E1 302.260} C_DIS
LIN {X -0.040,Y -297.802,Z 1675.666,A 0.000,B 0.000,C 90.000,E1 299.873} C_DIS
LIN {X -0.053,Y -315.116,Z 1675.653,A 0.000,B 0.000,C 90.000,E1 297.564} C_DIS
LIN {X -0.157,Y -327.670,Z 1675.644,A 0.000,B 0.000,C 90.000,E1 295.976} C_DIS
LIN {X -0.081,Y -342.536,Z 1675.634,A 0.000,B 0.000,C 90.000,E1 294.079} C_DIS
LIN {X 0.148,Y -357.560,Z 1675.624,A 0.000,B 0.000,C 90.000,E1 292.206} C_DIS
LIN {X -0.027,Y -369.773,Z 1675.615,A 0.000,B 0.000,C 90.000,E1 290.737} C_DIS
LIN {X -0.102,Y -376.667,Z 1675.610,A 0.000,B 0.000,C 90.000,E1 289.866} C_DIS
LIN {X 0.107,Y -383.110,Z 1675.605,A 0.000,B 0.000,C 90.000,E1 288.960} C_DIS
LIN {X -0.100,Y -388.888,Z 1675.601,A 0.000,B 0.000,C 90.000,E1 288.127} C_DIS
LIN {X 0.198,Y -392.283,Z 1675.597,A 0.000,B 0.000,C 90.000,E1 287.511} C_DIS
LIN {X 0.073,Y -396.605,Z 1675.593,A 0.000,B 0.000,C 90.000,E1 286.677} C_DIS
LIN {X -0.077,Y -398.995,Z 1675.590,A 0.000,B 0.000,C 90.000,E1 286.134} C_DIS
LIN {X 0.064,Y -400.987,Z 1675.586,A 0.000,B 0.000,C 90.000,E1 285.552} C_DIS
LIN {X -0.067,Y -402.648,Z 1675.583,A 0.000,B 0.000,C 90.000,E1 285.009} C_DIS
LIN {X 0.100,Y -403.945,Z 1675.580,A 0.000,B 0.000,C 90.000,E1 284.426} C_DIS
LIN {X -0.014,Y -404.822,Z 1675.577,A 0.000,B 0.000,C 90.000,E1 283.883} C_DIS
LIN {X 0.174,Y -405.318,Z 1675.574,A 0.000,B 0.000,C 90.000,E1 283.300} C_DIS
LIN {X -0.025,Y -405.380,Z 1675.571,A 0.000,B 0.000,C 90.000,E1 282.771} C_DIS
LIN {X -0.220,Y -404.994,Z 1675.568,A 0.000,B 0.000,C 90.000,E1 282.243} C_DIS
LIN {X -0.018,Y -404.115,Z 1675.565,A 0.000,B 0.000,C 90.000,E1 281.658} C_DIS
LIN {X -0.215,Y -402.694,Z 1675.562,A 0.000,B 0.000,C 90.000,E1 281.130} C_DIS
LIN {X -0.023,Y -400.763,Z 1675.559,A 0.000,B 0.000,C 90.000,E1 280.546} C_DIS
LIN {X 0.158,Y -398.215,Z 1675.555,A 0.000,B 0.000,C 90.000,E1 279.962} C_DIS
LIN {X -0.068,Y -393.437,Z 1675.551,A 0.000,B 0.000,C 90.000,E1 279.151} C_DIS
LIN {X 0.120,Y -387.858,Z 1675.546,A 0.000,B 0.000,C 90.000,E1 278.276} C_DIS
LIN {X 0.190,Y -381.620,Z 1675.541,A 0.000,B 0.000,C 90.000,E1 277.409} C_DIS
LIN {X 0.166,Y -374.245,Z 1675.536,A 0.000,B 0.000,C 90.000,E1 276.549} C_DIS
LIN {X 0.185,Y -368.496,Z 1675.533,A 0.000,B 0.000,C 90.000,E1 275.967} C_DIS
LIN {X 0.074,Y -362.577,Z 1675.530,A 0.000,B 0.000,C 90.000,E1 275.454} C_DIS
LIN {X -0.102,Y -356.357,Z 1675.528,A 0.000,B 0.000,C 90.000,E1 274.992} C_DIS
LIN {X 0.036,Y -350.018,Z 1675.525,A 0.000,B 0.000,C 90.000,E1 274.531} C_DIS
LIN {X 0.039,Y -340.199,Z 1675.522,A 0.000,B 0.000,C 90.000,E1 273.955} C_DIS
LIN {X 0.152,Y -330.577,Z 1675.519,A 0.000,B 0.000,C 90.000,E1 273.440} C_DIS
LIN {X -0.073,Y -320.944,Z 1675.517,A 0.000,B 0.000,C 90.000,E1 273.037} C_DIS
LIN {X -0.087,Y -310.999,Z 1675.515,A 0.000,B 0.000,C 90.000,E1 272.636} C_DIS
LIN {X -0.144,Y -300.860,Z 1675.513,A 0.000,B 0.000,C 90.000,E1 272.293} C_DIS
LIN {X 0.068,Y -289.826,Z 1675.511,A 0.000,B 0.000,C 90.000,E1 271.949} C_DIS
LIN {X 0.064,Y -277.957,Z 1675.510,A 0.000,B 0.000,C 90.000,E1 271.718} C_DIS
LIN {X -0.105,Y -265.455,Z 1675.509,A 0.000,B 0.000,C 90.000,E1 271.604} C_DIS
LIN {X -0.109,Y -250.645,Z 1675.508,A 0.000,B 0.000,C 90.000,E1 271.547} C_DIS
LIN {X 0.056,Y -205.171,Z 1675.508,A 0.000,B 0.000,C 90.000,E1 271.375} C_DIS
LIN {X 0.074,Y -182.450,Z 1675.507,A 0.000,B 0.000,C 90.000,E1 271.260} C_DIS
LIN {X 0.039,Y -181.397,Z 1675.507,A 0.000,B 0.000,C 90.000,E1 271.260} C_DIS
LIN {X 0.077,Y -181.581,Z 1675.501,A 0.000,B 0.000,C 90.000,E1 270.229} C_DIS
LIN {X 0.080,Y -180.869,Z 1675.472,A 0.000,B 0.000,C 90.000,E1 265.008} C_DIS
LIN {X -0.043,Y -178.984,Z 1675.444,A 0.000,B 0.000,C 90.000,E1 259.982} C_DIS
LIN {X -0.031,Y -177.960,Z 1675.435,A 0.000,B 0.000,C 90.000,E1 258.285} C_DIS
LIN {X -0.013,Y -175.603,Z 1675.411,A 0.000,B 0.000,C 90.000,E1 254.031} C_DIS
LIN {X 0.000,Y -172.326,Z 1675.388,A 0.000,B 0.000,C 90.000,E1 249.752} C_DIS
LIN {X -0.021,Y -171.803,Z 1675.383,A 0.000,B 0.000,C 90.000,E1 248.901} C_DIS
LIN {X 0.016,Y -169.478,Z 1675.368,A 0.000,B 0.000,C 90.000,E1 246.305} C_DIS
LIN {X -0.077,Y -166.805,Z 1675.349,A 0.000,B 0.000,C 90.000,E1 242.871} C_DIS
LIN {X 0.066,Y -162.786,Z 1675.325,A 0.000,B 0.000,C 90.000,E1 238.456} C_DIS
LIN {X 0.041,Y -161.474,Z 1675.315,A 0.000,B 0.000,C 90.000,E1 236.707} C_DIS
LIN {X 0.081,Y -157.469,Z 1675.291,A 0.000,B 0.000,C 90.000,E1 232.271} C_DIS
LIN {X 0.015,Y -155.484,Z 1675.276,A 0.000,B 0.000,C 90.000,E1 229.622} C_DIS
LIN {X -0.053,Y -151.792,Z 1675.251,A 0.000,B 0.000,C 90.000,E1 225.162} C_DIS
LIN {X -0.040,Y -150.000,Z 1675.236,A 0.000,B 0.000,C 90.000,E1 222.447} C_DIS
LIN {X -0.008,Y -146.829,Z 1675.210,A 0.000,B 0.000,C 90.000,E1 217.890} C_DIS
LIN {X -0.022,Y -145.409,Z 1675.195,A 0.000,B 0.000,C 90.000,E1 215.152} C_DIS
LIN {X 0.014,Y -142.840,Z 1675.170,A 0.000,B 0.000,C 90.000,E1 210.541} C_DIS
LIN {X -0.056,Y -141.454,Z 1675.149,A 0.000,B 0.000,C 90.000,E1 206.873} C_DIS
LIN {X -0.016,Y -139.373,Z 1675.113,A 0.000,B 0.000,C 90.000,E1 200.355} C_DIS
LIN {X -0.074,Y -138.821,Z 1675.098,A 0.000,B 0.000,C 90.000,E1 197.583} C_DIS
LIN {X 0.015,Y -138.353,Z 1675.056,A 0.000,B 0.000,C 90.000,E1 190.074} C_DIS
LIN {X -0.012,Y -139.533,Z 1675.004,A 0.000,B 0.000,C 90.000,E1 180.745} C_DIS
LIN {X -0.060,Y -141.216,Z 1674.973,A 0.000,B 0.000,C 90.000,E1 175.179} C_DIS
LIN {X 0.040,Y -142.589,Z 1674.958,A 0.000,B 0.000,C 90.000,E1 172.356} C_DIS
LIN {X -0.006,Y -144.888,Z 1674.932,A 0.000,B 0.000,C 90.000,E1 167.757} C_DIS
LIN {X -0.052,Y -147.517,Z 1674.912,A 0.000,B 0.000,C 90.000,E1 164.102} C_DIS
LIN {X 0.022,Y -150.111,Z 1674.891,A 0.000,B 0.000,C 90.000,E1 160.423} C_DIS
LIN {X 0.034,Y -153.470,Z 1674.871,A 0.000,B 0.000,C 90.000,E1 156.794} C_DIS
LIN {X 0.025,Y -157.834,Z 1674.846,A 0.000,B 0.000,C 90.000,E1 152.308} C_DIS
LIN {X 0.055,Y -162.117,Z 1674.826,A 0.000,B 0.000,C 90.000,E1 148.742} C_DIS
LIN {X -0.060,Y -166.320,Z 1674.807,A 0.000,B 0.000,C 90.000,E1 145.261} C_DIS
LIN {X 0.042,Y -171.337,Z 1674.788,A 0.000,B 0.000,C 90.000,E1 141.743} C_DIS
LIN {X -0.030,Y -176.239,Z 1674.768,A 0.000,B 0.000,C 90.000,E1 138.324} C_DIS
LIN {X 0.089,Y -180.520,Z 1674.754,A 0.000,B 0.000,C 90.000,E1 135.729} C_DIS
LIN {X 0.069,Y -185.923,Z 1674.735,A 0.000,B 0.000,C 90.000,E1 132.366} C_DIS
LIN {X 0.004,Y -190.551,Z 1674.722,A 0.000,B 0.000,C 90.000,E1 129.886} C_DIS
LIN {X 0.034,Y -196.302,Z 1674.703,A 0.000,B 0.000,C 90.000,E1 126.583} C_DIS
LIN {X 0.112,Y -201.102,Z 1674.690,A 0.000,B 0.000,C 90.000,E1 124.119} C_DIS
LIN {X 0.022,Y -207.400,Z 1674.671,A 0.000,B 0.000,C 90.000,E1 120.747} C_DIS
LIN {X 0.104,Y -207.934,Z 1674.669,A 0.000,B 0.000,C 90.000,E1 120.463} C_DIS
LIN {X 0.111,Y -330.315,Z 1674.669,A 0.000,B 0.000,C 90.000,E1 120.463} C_DIS
LIN {X 0.004,Y -331.424,Z 1674.669,A 0.000,B 0.000,C 90.000,E1 120.463} C_DIS
LIN {X -0.206,Y -335.540,Z 1674.668,A 0.000,B 0.000,C 90.000,E1 120.335} C_DIS
LIN {X 0.042,Y -337.859,Z 1674.667,A 0.000,B 0.000,C 90.000,E1 120.129} C_DIS
LIN {X -0.159,Y -341.723,Z 1674.665,A 0.000,B 0.000,C 90.000,E1 119.745} C_DIS
LIN {X 0.098,Y -343.592,Z 1674.663,A 0.000,B 0.000,C 90.000,E1 119.411} C_DIS
LIN {X 0.052,Y -346.377,Z 1674.660,A 0.000,B 0.000,C 90.000,E1 118.821} C_DIS
LIN {X -0.045,Y -359.022,Z 1674.645,A 0.000,B 0.000,C 90.000,E1 116.104} C_DIS
LIN {X -0.108,Y -373.167,Z 1674.630,A 0.000,B 0.000,C 90.000,E1 113.439} C_DIS
LIN {X -0.014,Y -387.102,Z 1674.617,A 0.000,B 0.000,C 90.000,E1 111.099} C_DIS
LIN {X -0.072,Y -402.416,Z 1674.605,A 0.000,B 0.000,C 90.000,E1 108.833} C_DIS
LIN {X -0.142,Y -419.215,Z 1674.592,A 0.000,B 0.000,C 90.000,E1 106.622} C_DIS
LIN {X 0.105,Y -437.616,Z 1674.580,A 0.000,B 0.000,C 90.000,E1 104.426} C_DIS
LIN {X 0.124,Y -457.377,Z 1674.569,A 0.000,B 0.000,C 90.000,E1 102.355} C_DIS
LIN {X -0.194,Y -477.736,Z 1674.558,A 0.000,B 0.000,C 90.000,E1 100.489} C_DIS
LIN {X -0.060,Y -501.248,Z 1674.547,A 0.000,B 0.000,C 90.000,E1 98.511} C_DIS
LIN {X 0.172,Y -503.507,Z 1674.546,A 0.000,B 0.000,C 90.000,E1 98.276} C_DIS
LIN {X -0.165,Y -505.220,Z 1674.545,A 0.000,B 0.000,C 90.000,E1 98.106} C_DIS
LIN {X 0.273,Y -506.737,Z 1674.544,A 0.000,B 0.000,C 90.000,E1 97.814} C_DIS
LIN {X 0.143,Y -507.864,Z 1674.542,A 0.000,B 0.000,C 90.000,E1 97.587} C_DIS
LIN {X -0.034,Y -509.184,Z 1674.540,A 0.000,B 0.000,C 90.000,E1 97.125} C_DIS
LIN {X -0.204,Y -509.446,Z 1674.537,A 0.000,B 0.000,C 90.000,E1 96.663} C_DIS
LIN {X 0.140,Y -508.694,Z 1674.534,A 0.000,B 0.000,C 90.000,E1 96.144} C_DIS
LIN {X -0.022,Y -506.798,Z 1674.531,A 0.000,B 0.000,C 90.000,E1 95.682} C_DIS
LIN {X -0.130,Y -505.301,Z 1674.530,A 0.000,B 0.000,C 90.000,E1 95.454} C_DIS
LIN {X 0.149,Y -493.066,Z 1674.521,A 0.000,B 0.000,C 90.000,E1 93.726} C_DIS
LIN {X 0.111,Y -480.604,Z 1674.511,A 0.000,B 0.000,C 90.000,E1 92.007} C_DIS
LIN {X -0.159,Y -467.984,Z 1674.501,A 0.000,B 0.000,C 90.000,E1 90.286} C_DIS
LIN {X 0.002,Y -457.140,Z 1674.493,A 0.000,B 0.000,C 90.000,E1 88.740} C_DIS
LIN {X -0.021,Y -446.029,Z 1674.484,A 0.000,B 0.000,C 90.000,E1 87.192} C_DIS
LIN {X -0.203,Y -434.561,Z 1674.476,A 0.000,B 0.000,C 90.000,E1 85.641} C_DIS
LIN {X 0.002,Y -421.197,Z 1674.465,A 0.000,B 0.000,C 90.000,E1 83.742} C_DIS
LIN {X 0.200,Y -404.448,Z 1674.452,A 0.000,B 0.000,C 90.000,E1 81.254} C_DIS
LIN {X 0.068,Y -386.869,Z 1674.436,A 0.000,B 0.000,C 90.000,E1 78.465} C_DIS
LIN {X 0.021,Y -371.687,Z 1674.422,A 0.000,B 0.000,C 90.000,E1 75.880} C_DIS
LIN {X 0.209,Y -357.123,Z 1674.407,A 0.000,B 0.000,C 90.000,E1 73.196} C_DIS
LIN {X 0.121,Y -340.181,Z 1674.388,A 0.000,B 0.000,C 90.000,E1 69.880} C_DIS
LIN {X 0.053,Y -328.697,Z 1674.375,A 0.000,B 0.000,C 90.000,E1 67.411} C_DIS
LIN {X -0.162,Y -317.651,Z 1674.360,A 0.000,B 0.000,C 90.000,E1 64.921} C_DIS
LIN {X 0.075,Y -305.482,Z 1674.344,A 0.000,B 0.000,C 90.000,E1 61.975} C_DIS
LIN {X 0.099,Y -297.354,Z 1674.333,A 0.000,B 0.000,C 90.000,E1 59.999} C_DIS
LIN {X 0.120,Y -289.028,Z 1674.322,A 0.000,B 0.000,C 90.000,E1 57.995} C_DIS
LIN {X -0.098,Y -280.436,Z 1674.311,A 0.000,B 0.000,C 90.000,E1 56.008} C_DIS
LIN {X 0.000,Y -270.316,Z 1674.298,A 0.000,B 0.000,C 90.000,E1 53.577} C_DIS
LIN {X -0.123,Y -257.556,Z 1674.280,A 0.000,B 0.000,C 90.000,E1 50.436} C_DIS
LIN {X 0.060,Y -245.561,Z 1674.262,A 0.000,B 0.000,C 90.000,E1 47.148} C_DIS
LIN {X -0.107,Y -234.553,Z 1674.244,A 0.000,B 0.000,C 90.000,E1 43.866} C_DIS
LIN {X -0.004,Y -225.639,Z 1674.227,A 0.000,B 0.000,C 90.000,E1 40.825} C_DIS
LIN {X 0.116,Y -217.495,Z 1674.210,A 0.000,B 0.000,C 90.000,E1 37.729} C_DIS
LIN {X 0.116,Y -210.005,Z 1674.193,A 0.000,B 0.000,C 90.000,E1 34.612} C_DIS
LIN {X 0.044,Y -203.098,Z 1674.175,A 0.000,B 0.000,C 90.000,E1 31.465} C_DIS
LIN {X -0.062,Y -196.688,Z 1674.157,A 0.000,B 0.000,C 90.000,E1 28.281} C_DIS
LIN {X -0.077,Y -190.880,Z 1674.139,A 0.000,B 0.000,C 90.000,E1 25.027} C_DIS
LIN {X -0.043,Y -185.653,Z 1674.121,A 0.000,B 0.000,C 90.000,E1 21.716} C_DIS
LIN {X 0.002,Y -180.984,Z 1674.102,A 0.000,B 0.000,C 90.000,E1 18.362} C_DIS
LIN {X -0.065,Y -177.025,Z 1674.083,A 0.000,B 0.000,C 90.000,E1 15.009} C_DIS
LIN {X 0.037,Y -173.118,Z 1674.060,A 0.000,B 0.000,C 90.000,E1 10.715} C_DIS
LIN {X -0.006,Y -169.774,Z 1674.031,A 0.000,B 0.000,C 90.000,E1 5.568} C_DIS
LIN {X -0.030,Y -167.460,Z 1673.997,A 0.000,B 0.000,C 90.000,E1 359.542} C_DIS
LIN {X -0.018,Y -168.329,Z 1673.930,A 0.000,B 0.000,C 90.000,E1 347.353} C_DIS
LIN {X 0.058,Y -171.041,Z 1673.901,A 0.000,B 0.000,C 90.000,E1 342.127} C_DIS
LIN {X -0.022,Y -174.505,Z 1673.877,A 0.000,B 0.000,C 90.000,E1 337.847} C_DIS
LIN {X 0.040,Y -178.265,Z 1673.858,A 0.000,B 0.000,C 90.000,E1 334.409} C_DIS
LIN {X -0.056,Y -182.735,Z 1673.839,A 0.000,B 0.000,C 90.000,E1 331.051} C_DIS
LIN {X 0.066,Y -188.103,Z 1673.820,A 0.000,B 0.000,C 90.000,E1 327.661} C_DIS
LIN {X 0.038,Y -192.763,Z 1673.807,A 0.000,B 0.000,C 90.000,E1 325.182} C_DIS
LIN {X 0.047,Y -198.084,Z 1673.793,A 0.000,B 0.000,C 90.000,E1 322.718} C_DIS
LIN {X -0.031,Y -205.130,Z 1673.777,A 0.000,B 0.000,C 90.000,E1 319.908} C_DIS
LIN {X 0.031,Y -213.058,Z 1673.762,A 0.000,B 0.000,C 90.000,E1 317.106} C_DIS
LIN {X 0.035,Y -220.712,Z 1673.749,A 0.000,B 0.000,C 90.000,E1 314.757} C_DIS
LIN {X 0.074,Y -232.076,Z 1673.732,A 0.000,B 0.000,C 90.000,E1 311.676} C_DIS
LIN {X 0.004,Y -241.606,Z 1673.719,A 0.000,B 0.000,C 90.000,E1 309.439} C_DIS
LIN {X -0.042,Y -250.389,Z 1673.709,A 0.000,B 0.000,C 90.000,E1 307.604} C_DIS
LIN {X 0.079,Y -266.130,Z 1673.693,A 0.000,B 0.000,C 90.000,E1 304.692} C_DIS
LIN {X -0.022,Y -281.362,Z 1673.679,A 0.000,B 0.000,C 90.000,E1 302.260} C_DIS
LIN {X 0.014,Y -297.864,Z 1673.666,A 0.000,B 0.000,C 90.000,E1 299.873} C_DIS
LIN {X -0.140,Y -315.183,Z 1673.653,A 0.000,B 0.000,C 90.000,E1 297.590} C_DIS
LIN {X -0.095,Y -327.745,Z 1673.644,A 0.000,B 0.000,C 90.000,E1 295.976} C_DIS
LIN {X -0.014,Y -342.584,Z 1673.634,A 0.000,B 0.000,C 90.000,E1 294.079} C_DIS
LIN {X 0.217,Y -357.574,Z 1673.624,A 0.000,B 0.000,C 90.000,E1 292.206} C_DIS
LIN {X 0.046,Y -369.752,Z 1673.615,A 0.000,B 0.000,C 90.000,E1 290.737} C_DIS
LIN {X -0.028,Y -376.631,Z 1673.610,A 0.000,B 0.000,C 90.000,E1 289.866} C_DIS
LIN {X 0.182,Y -383.088,Z 1673.605,A 0.000,B 0.000,C 90.000,E1 288.960} C_DIS
LIN {X -0.024,Y -388.874,Z 1673.601,A 0.000,B 0.000,C 90.000,E1 288.127} C_DIS
LIN {X -0.218,Y -392.301,Z 1673.598,A 0.000,B 0.000,C 90.000,E1 287.583} C_DIS
LIN {X 0.150,Y -396.634,Z 1673.593,A 0.000,B 0.000,C 90.000,E1 286.677} C_DIS
LIN {X 0.001,Y -399.023,Z 1673.590,A 0.000,B 0.000,C 90.000,E1 286.134} C_DIS
LIN {X 0.142,Y -401.048,Z 1673.587,A 0.000,B 0.000,C 90.000,E1 285.552} C_DIS
LIN {X 0.012,Y -402.719,Z 1673.583,A 0.000,B 0.000,C 90.000,E1 285.009} C_DIS
LIN {X -0.212,Y -404.026,Z 1673.580,A 0.000,B 0.000,C 90.000,E1 284.481} C_DIS
LIN {X 0.066,Y -404.960,Z 1673.577,A 0.000,B 0.000,C 90.000,E1 283.883} C_DIS
LIN {X -0.139,Y -405.436,Z 1673.574,A 0.000,B 0.000,C 90.000,E1 283.355} C_DIS
LIN {X 0.057,Y -405.506,Z 1673.571,A 0.000,B 0.000,C 90.000,E1 282.771} C_DIS
LIN {X -0.138,Y -405.117,Z 1673.568,A 0.000,B 0.000,C 90.000,E1 282.243} C_DIS
LIN {X 0.065,Y -404.270,Z 1673.565,A 0.000,B 0.000,C 90.000,E1 281.658} C_DIS
LIN {X -0.132,Y -402.867,Z 1673.562,A 0.000,B 0.000,C 90.000,E1 281.130} C_DIS
LIN {X 0.061,Y -400.941,Z 1673.559,A 0.000,B 0.000,C 90.000,E1 280.546} C_DIS
LIN {X -0.150,Y -398.420,Z 1673.556,A 0.000,B 0.000,C 90.000,E1 280.018} C_DIS
LIN {X -0.054,Y -395.322,Z 1673.552,A 0.000,B 0.000,C 90.000,E1 279.443} C_DIS
LIN {X 0.149,Y -390.002,Z 1673.548,A 0.000,B 0.000,C 90.000,E1 278.568} C_DIS
LIN {X -0.136,Y -383.922,Z 1673.543,A 0.000,B 0.000,C 90.000,E1 277.757} C_DIS
LIN {X -0.115,Y -379.385,Z 1673.540,A 0.000,B 0.000,C 90.000,E1 277.182} C_DIS
LIN {X -0.120,Y -374.306,Z 1673.537,A 0.000,B 0.000,C 90.000,E1 276.606} C_DIS
LIN {X -0.102,Y -368.618,Z 1673.533,A 0.000,B 0.000,C 90.000,E1 276.030} C_DIS
LIN {X -0.148,Y -362.705,Z 1673.531,A 0.000,B 0.000,C 90.000,E1 275.511} C_DIS
LIN {X 0.064,Y -356.554,Z 1673.528,A 0.000,B 0.000,C 90.000,E1 274.992} C_DIS
LIN {X 0.178,Y -350.058,Z 1673.525,A 0.000,B 0.000,C 90.000,E1 274.531} C_DIS
LIN {X -0.142,Y -343.428,Z 1673.523,A 0.000,B 0.000,C 90.000,E1 274.188} C_DIS
LIN {X -0.102,Y -333.838,Z 1673.520,A 0.000,B 0.000,C 90.000,E1 273.669} C_DIS
LIN {X -0.159,Y -324.062,Z 1673.518,A 0.000,B 0.000,C 90.000,E1 273.212} C_DIS
LIN {X 0.072,Y -314.156,Z 1673.515,A 0.000,B 0.000,C 90.000,E1 272.751} C_DIS
LIN {X -0.115,Y -303.971,Z 1673.513,A 0.000,B 0.000,C 90.000,E1 272.407} C_DIS
LIN {X -0.094,Y -296.696,Z 1673.512,A 0.000,B 0.000,C 90.000,E1 272.178} C_DIS
LIN {X 0.007,Y -285.550,Z 1673.510,A 0.000,B 0.000,C 90.000,E1 271.892} C_DIS
LIN {X -0.134,Y -277.384,Z 1673.510,A 0.000,B 0.000,C 90.000,E1 271.776} C_DIS
LIN {X -0.020,Y -264.456,Z 1673.509,A 0.000,B 0.000,C 90.000,E1 271.604} C_DIS
LIN {X 0.047,Y -235.176,Z 1673.508,A 0.000,B 0.000,C 90.000,E1 271.489} C_DIS
LIN {X -0.022,Y -197.919,Z 1673.508,A 0.000,B 0.000,C 90.000,E1 271.375} C_DIS
LIN {X -0.069,Y -182.785,Z 1673.507,A 0.000,B 0.000,C 90.000,E1 271.318} C_DIS
LIN {X -0.087,Y -181.393,Z 1673.507,A 0.000,B 0.000,C 90.000,E1 271.318} C_DIS
LIN {X -0.073,Y -181.581,Z 1673.501,A 0.000,B 0.000,C 90.000,E1 270.286} C_DIS
LIN {X -0.068,Y -180.871,Z 1673.472,A 0.000,B 0.000,C 90.000,E1 265.065} C_DIS
LIN {X -0.011,Y -178.987,Z 1673.444,A 0.000,B 0.000,C 90.000,E1 259.982} C_DIS
LIN {X 0.001,Y -177.968,Z 1673.435,A 0.000,B 0.000,C 90.000,E1 258.285} C_DIS
LIN {X 0.019,Y -175.610,Z 1673.411,A 0.000,B 0.000,C 90.000,E1 254.031} C_DIS
LIN {X 0.031,Y -172.332,Z 1673.388,A 0.000,B 0.000,C 90.000,E1 249.752} C_DIS
LIN {X 0.010,Y -171.810,Z 1673.383,A 0.000,B 0.000,C 90.000,E1 248.901} C_DIS
LIN {X 0.018,Y -170.271,Z 1673.373,A 0.000,B 0.000,C 90.000,E1 247.177} C_DIS
LIN {X -0.046,Y -166.813,Z 1673.349,A 0.000,B 0.000,C 90.000,E1 242.871} C_DIS
LIN {X 0.011,Y -162.795,Z 1673.325,A 0.000,B 0.000,C 90.000,E1 238.486} C_DIS
LIN {X 0.072,Y -161.483,Z 1673.315,A 0.000,B 0.000,C 90.000,E1 236.707} C_DIS
LIN {X -0.012,Y -157.478,Z 1673.291,A 0.000,B 0.000,C 90.000,E1 232.316} C_DIS
LIN {X 0.044,Y -155.494,Z 1673.276,A 0.000,B 0.000,C 90.000,E1 229.622} C_DIS
LIN {X -0.024,Y -151.799,Z 1673.251,A 0.000,B 0.000,C 90.000,E1 225.162} C_DIS
LIN {X -0.010,Y -150.009,Z 1673.236,A 0.000,B 0.000,C 90.000,E1 222.447} C_DIS
LIN {X 0.020,Y -146.836,Z 1673.211,A 0.000,B 0.000,C 90.000,E1 217.890} C_DIS
LIN {X 0.007,Y -145.416,Z 1673.195,A 0.000,B 0.000,C 90.000,E1 215.152} C_DIS
LIN {X 0.042,Y -142.845,Z 1673.170,A 0.000,B 0.000,C 90.000,E1 210.541} C_DIS
LIN {X -0.028,Y -141.459,Z 1673.149,A 0.000,B 0.000,C 90.000,E1 206.873} C_DIS
LIN {X 0.011,Y -139.374,Z 1673.113,A 0.000,B 0.000,C 90.000,E1 200.355} C_DIS
LIN {X -0.047,Y -138.825,Z 1673.098,A 0.000,B 0.000,C 90.000,E1 197.583} C_DIS
LIN {X 0.042,Y -138.353,Z 1673.056,A 0.000,B 0.000,C 90.000,E1 190.074} C_DIS
LIN {X 0.016,Y -139.531,Z 1673.004,A 0.000,B 0.000,C 90.000,E1 180.745} C_DIS
LIN {X -0.032,Y -141.210,Z 1672.973,A 0.000,B 0.000,C 90.000,E1 175.179} C_DIS
LIN {X 0.069,Y -142.585,Z 1672.958,A 0.000,B 0.000,C 90.000,E1 172.356} C_DIS
LIN {X 0.023,Y -144.882,Z 1672.932,A 0.000,B 0.000,C 90.000,E1 167.757} C_DIS
LIN {X -0.024,Y -147.509,Z 1672.912,A 0.000,B 0.000,C 90.000,E1 164.102} C_DIS
LIN {X 0.051,Y -150.102,Z 1672.891,A 0.000,B 0.000,C 90.000,E1 160.423} C_DIS
LIN {X 0.064,Y -153.459,Z 1672.871,A 0.000,B 0.000,C 90.000,E1 156.794} C_DIS
LIN {X -0.085,Y -157.822,Z 1672.846,A 0.000,B 0.000,C 90.000,E1 152.359} C_DIS
LIN {X -0.053,Y -162.105,Z 1672.827,A 0.000,B 0.000,C 90.000,E1 148.791} C_DIS
LIN {X -0.029,Y -166.306,Z 1672.807,A 0.000,B 0.000,C 90.000,E1 145.261} C_DIS
LIN {X -0.033,Y -171.323,Z 1672.788,A 0.000,B 0.000,C 90.000,E1 141.778} C_DIS
LIN {X 0.002,Y -176.223,Z 1672.768,A 0.000,B 0.000,C 90.000,E1 138.324} C_DIS
LIN {X -0.004,Y -180.502,Z 1672.754,A 0.000,B 0.000,C 90.000,E1 135.769} C_DIS
LIN {X -0.023,Y -185.904,Z 1672.736,A 0.000,B 0.000,C 90.000,E1 132.405} C_DIS
LIN {X 0.038,Y -190.533,Z 1672.722,A 0.000,B 0.000,C 90.000,E1 129.886} C_DIS
LIN {X 0.069,Y -196.283,Z 1672.703,A 0.000,B 0.000,C 90.000,E1 126.583} C_DIS
LIN {X -0.131,Y -201.085,Z 1672.690,A 0.000,B 0.000,C 90.000,E1 124.199} C_DIS
LIN {X 0.057,Y -207.380,Z 1672.671,A 0.000,B 0.000,C 90.000,E1 120.747} C_DIS
LIN {X -0.035,Y -207.852,Z 1672.670,A 0.000,B 0.000,C 90.000,E1 120.541} C_DIS
LIN {X -0.116,Y -330.155,Z 1672.670,A 0.000,B 0.000,C 90.000,E1 120.541} C_DIS
LIN {X -0.039,Y -335.525,Z 1672.668,A 0.000,B 0.000,C 90.000,E1 120.335} C_DIS
LIN {X 0.100,Y -338.008,Z 1672.667,A 0.000,B 0.000,C 90.000,E1 120.129} C_DIS
LIN {X -0.016,Y -341.841,Z 1672.665,A 0.000,B 0.000,C 90.000,E1 119.716} C_DIS
LIN {X 0.020,Y -343.689,Z 1672.663,A 0.000,B 0.000,C 90.000,E1 119.411} C_DIS
LIN {X 0.086,Y -347.785,Z 1672.658,A 0.000,B 0.000,C 90.000,E1 118.487} C_DIS
LIN {X 0.030,Y -360.599,Z 1672.643,A 0.000,B 0.000,C 90.000,E1 115.771} C_DIS
LIN {X 0.195,Y -374.934,Z 1672.628,A 0.000,B 0.000,C 90.000,E1 113.078} C_DIS
LIN {X -0.010,Y -389.048,Z 1672.615,A 0.000,B 0.000,C 90.000,E1 110.791} C_DIS
LIN {X -0.153,Y -404.555,Z 1672.603,A 0.000,B 0.000,C 90.000,E1 108.544} C_DIS
LIN {X -0.042,Y -421.562,Z 1672.591,A 0.000,B 0.000,C 90.000,E1 106.315} C_DIS
LIN {X -0.169,Y -440.187,Z 1672.579,A 0.000,B 0.000,C 90.000,E1 104.175} C_DIS
LIN {X -0.115,Y -460.059,Z 1672.567,A 0.000,B 0.000,C 90.000,E1 102.119} C_DIS
LIN {X -0.166,Y -483.065,Z 1672.556,A 0.000,B 0.000,C 90.000,E1 100.018} C_DIS
LIN {X -0.193,Y -501.400,Z 1672.547,A 0.000,B 0.000,C 90.000,E1 98.511} C_DIS
LIN {X 0.194,Y -505.229,Z 1672.545,A 0.000,B 0.000,C 90.000,E1 98.049} C_DIS
LIN {X 0.126,Y -506.699,Z 1672.543,A 0.000,B 0.000,C 90.000,E1 97.814} C_DIS
LIN {X -0.011,Y -507.786,Z 1672.542,A 0.000,B 0.000,C 90.000,E1 97.587} C_DIS
LIN {X -0.188,Y -509.037,Z 1672.539,A 0.000,B 0.000,C 90.000,E1 97.125} C_DIS
LIN {X 0.147,Y -509.237,Z 1672.537,A 0.000,B 0.000,C 90.000,E1 96.606} C_DIS
LIN {X -0.016,Y -508.422,Z 1672.534,A 0.000,B 0.000,C 90.000,E1 96.144} C_DIS
LIN {X -0.178,Y -506.446,Z 1672.531,A 0.000,B 0.000,C 90.000,E1 95.682} C_DIS
LIN {X 0.156,Y -503.130,Z 1672.529,A 0.000,B 0.000,C 90.000,E1 95.163} C_DIS
LIN {X -0.150,Y -490.894,Z 1672.519,A 0.000,B 0.000,C 90.000,E1 93.498} C_DIS
LIN {X -0.199,Y -478.412,Z 1672.510,A 0.000,B 0.000,C 90.000,E1 91.776} C_DIS
LIN {X -0.056,Y -465.794,Z 1672.500,A 0.000,B 0.000,C 90.000,E1 90.000} C_DIS
LIN {X -0.161,Y -453.082,Z 1672.490,A 0.000,B 0.000,C 90.000,E1 88.224} C_DIS
LIN {X -0.001,Y -443.738,Z 1672.483,A 0.000,B 0.000,C 90.000,E1 86.906} C_DIS
LIN {X -0.041,Y -430.296,Z 1672.473,A 0.000,B 0.000,C 90.000,E1 85.065} C_DIS
LIN {X 0.072,Y -416.949,Z 1672.462,A 0.000,B 0.000,C 90.000,E1 83.166} C_DIS
LIN {X 0.153,Y -400.370,Z 1672.448,A 0.000,B 0.000,C 90.000,E1 80.679} C_DIS
LIN {X -0.075,Y -384.699,Z 1672.434,A 0.000,B 0.000,C 90.000,E1 78.173} C_DIS
LIN {X -0.079,Y -369.590,Z 1672.420,A 0.000,B 0.000,C 90.000,E1 75.574} C_DIS
LIN {X -0.041,Y -355.065,Z 1672.405,A 0.000,B 0.000,C 90.000,E1 72.906} C_DIS
LIN {X -0.074,Y -338.296,Z 1672.386,A 0.000,B 0.000,C 90.000,E1 69.571} C_DIS
LIN {X 0.121,Y -326.843,Z 1672.373,A 0.000,B 0.000,C 90.000,E1 67.050} C_DIS
LIN {X -0.013,Y -315.838,Z 1672.359,A 0.000,B 0.000,C 90.000,E1 64.537} C_DIS
LIN {X -0.139,Y -305.052,Z 1672.344,A 0.000,B 0.000,C 90.000,E1 61.975} C_DIS
LIN {X -0.117,Y -296.920,Z 1672.333,A 0.000,B 0.000,C 90.000,E1 59.999} C_DIS
LIN {X -0.092,Y -289.978,Z 1672.324,A 0.000,B 0.000,C 90.000,E1 58.329} C_DIS
LIN {X -0.053,Y -281.417,Z 1672.313,A 0.000,B 0.000,C 90.000,E1 56.294} C_DIS
LIN {X -0.063,Y -269.822,Z 1672.297,A 0.000,B 0.000,C 90.000,E1 53.543} C_DIS
LIN {X 0.013,Y -257.081,Z 1672.280,A 0.000,B 0.000,C 90.000,E1 50.356} C_DIS
LIN {X 0.012,Y -245.171,Z 1672.262,A 0.000,B 0.000,C 90.000,E1 47.106} C_DIS
LIN {X -0.003,Y -234.243,Z 1672.243,A 0.000,B 0.000,C 90.000,E1 43.785} C_DIS
LIN {X -0.059,Y -225.374,Z 1672.226,A 0.000,B 0.000,C 90.000,E1 40.782} C_DIS
LIN {X -0.109,Y -217.235,Z 1672.209,A 0.000,B 0.000,C 90.000,E1 37.729} C_DIS
LIN {X -0.107,Y -209.763,Z 1672.192,A 0.000,B 0.000,C 90.000,E1 34.612} C_DIS
LIN {X -0.005,Y -202.851,Z 1672.175,A 0.000,B 0.000,C 90.000,E1 31.416} C_DIS
LIN {X -0.109,Y -196.448,Z 1672.157,A 0.000,B 0.000,C 90.000,E1 28.231} C_DIS
LIN {X -0.043,Y -190.642,Z 1672.139,A 0.000,B 0.000,C 90.000,E1 24.951} C_DIS
LIN {X -0.022,Y -185.446,Z 1672.120,A 0.000,B 0.000,C 90.000,E1 21.642} C_DIS
LIN {X -0.045,Y -180.809,Z 1672.102,A 0.000,B 0.000,C 90.000,E1 18.308} C_DIS
LIN {X 0.058,Y -176.886,Z 1672.083,A 0.000,B 0.000,C 90.000,E1 14.898} C_DIS
LIN {X -0.011,Y -173.020,Z 1672.059,A 0.000,B 0.000,C 90.000,E1 10.658} C_DIS
LIN {X -0.052,Y -169.719,Z 1672.031,A 0.000,B 0.000,C 90.000,E1 5.511} C_DIS
LIN {X -0.030,Y -167.466,Z 1671.997,A 0.000,B 0.000,C 90.000,E1 359.542} C_DIS
LIN {X -0.017,Y -168.329,Z 1671.930,A 0.000,B 0.000,C 90.000,E1 347.353} C_DIS
LIN {X 0.059,Y -171.063,Z 1671.901,A 0.000,B 0.000,C 90.000,E1 342.127} C_DIS
LIN {X -0.021,Y -174.552,Z 1671.877,A 0.000,B 0.000,C 90.000,E1 337.847} C_DIS
LIN {X 0.042,Y -178.336,Z 1671.858,A 0.000,B 0.000,C 90.000,E1 334.409} C_DIS
LIN {X -0.052,Y -182.840,Z 1671.839,A 0.000,B 0.000,C 90.000,E1 331.051} C_DIS
LIN {X 0.073,Y -188.220,Z 1671.820,A 0.000,B 0.000,C 90.000,E1 327.661} C_DIS
LIN {X 0.048,Y -192.920,Z 1671.807,A 0.000,B 0.000,C 90.000,E1 325.182} C_DIS
LIN {X -0.097,Y -198.243,Z 1671.793,A 0.000,B 0.000,C 90.000,E1 322.763} C_DIS
LIN {X -0.014,Y -205.313,Z 1671.777,A 0.000,B 0.000,C 90.000,E1 319.908} C_DIS
LIN {X -0.060,Y -214.448,Z 1671.760,A 0.000,B 0.000,C 90.000,E1 316.743} C_DIS
LIN {X -0.113,Y -223.614,Z 1671.744,A 0.000,B 0.000,C 90.000,E1 314.028} C_DIS
LIN {X 0.060,Y -233.761,Z 1671.730,A 0.000,B 0.000,C 90.000,E1 311.310} C_DIS
LIN {X 0.024,Y -243.439,Z 1671.717,A 0.000,B 0.000,C 90.000,E1 309.072} C_DIS
LIN {X 0.003,Y -252.385,Z 1671.707,A 0.000,B 0.000,C 90.000,E1 307.237} C_DIS
LIN {X 0.026,Y -268.328,Z 1671.691,A 0.000,B 0.000,C 90.000,E1 304.358} C_DIS
LIN {X 0.030,Y -281.465,Z 1671.679,A 0.000,B 0.000,C 90.000,E1 302.260} C_DIS
LIN {X 0.071,Y -297.923,Z 1671.666,A 0.000,B 0.000,C 90.000,E1 299.873} C_DIS
LIN {X -0.079,Y -315.284,Z 1671.653,A 0.000,B 0.000,C 90.000,E1 297.590} C_DIS
LIN {X -0.031,Y -327.823,Z 1671.644,A 0.000,B 0.000,C 90.000,E1 295.976} C_DIS
LIN {X 0.055,Y -342.630,Z 1671.634,A 0.000,B 0.000,C 90.000,E1 294.079} C_DIS
LIN {X -0.041,Y -357.571,Z 1671.624,A 0.000,B 0.000,C 90.000,E1 292.259} C_DIS
LIN {X 0.121,Y -369.730,Z 1671.615,A 0.000,B 0.000,C 90.000,E1 290.737} C_DIS
LIN {X -0.079,Y -376.621,Z 1671.610,A 0.000,B 0.000,C 90.000,E1 289.885} C_DIS
LIN {X -0.103,Y -383.033,Z 1671.606,A 0.000,B 0.000,C 90.000,E1 289.014} C_DIS
LIN {X 0.054,Y -388.856,Z 1671.601,A 0.000,B 0.000,C 90.000,E1 288.127} C_DIS
LIN {X -0.139,Y -392.306,Z 1671.598,A 0.000,B 0.000,C 90.000,E1 287.583} C_DIS
LIN {X -0.150,Y -396.655,Z 1671.593,A 0.000,B 0.000,C 90.000,E1 286.732} C_DIS
LIN {X 0.152,Y -400.158,Z 1671.588,A 0.000,B 0.000,C 90.000,E1 285.843} C_DIS
LIN {X 0.101,Y -402.814,Z 1671.583,A 0.000,B 0.000,C 90.000,E1 285.009} C_DIS
LIN {X -0.122,Y -404.142,Z 1671.580,A 0.000,B 0.000,C 90.000,E1 284.481} C_DIS
LIN {X 0.156,Y -405.063,Z 1671.577,A 0.000,B 0.000,C 90.000,E1 283.883} C_DIS
LIN {X -0.049,Y -405.561,Z 1671.574,A 0.000,B 0.000,C 90.000,E1 283.355} C_DIS
LIN {X 0.149,Y -405.633,Z 1671.571,A 0.000,B 0.000,C 90.000,E1 282.771} C_DIS
LIN {X -0.045,Y -405.277,Z 1671.568,A 0.000,B 0.000,C 90.000,E1 282.243} C_DIS
LIN {X 0.157,Y -404.446,Z 1671.565,A 0.000,B 0.000,C 90.000,E1 281.658} C_DIS
LIN {X -0.039,Y -403.063,Z 1671.562,A 0.000,B 0.000,C 90.000,E1 281.130} C_DIS
LIN {X 0.155,Y -401.166,Z 1671.559,A 0.000,B 0.000,C 90.000,E1 280.546} C_DIS
LIN {X -0.056,Y -398.645,Z 1671.556,A 0.000,B 0.000,C 90.000,E1 280.018} C_DIS
LIN {X 0.113,Y -393.865,Z 1671.551,A 0.000,B 0.000,C 90.000,E1 279.151} C_DIS
LIN {X -0.138,Y -388.216,Z 1671.546,A 0.000,B 0.000,C 90.000,E1 278.341} C_DIS
LIN {X -0.006,Y -381.868,Z 1671.542,A 0.000,B 0.000,C 90.000,E1 277.466} C_DIS
LIN {X -0.025,Y -374.392,Z 1671.537,A 0.000,B 0.000,C 90.000,E1 276.606} C_DIS
LIN {X 0.005,Y -368.714,Z 1671.533,A 0.000,B 0.000,C 90.000,E1 276.030} C_DIS
LIN {X 0.031,Y -362.887,Z 1671.531,A 0.000,B 0.000,C 90.000,E1 275.511} C_DIS
LIN {X -0.080,Y -356.807,Z 1671.528,A 0.000,B 0.000,C 90.000,E1 275.049} C_DIS
LIN {X 0.057,Y -350.315,Z 1671.526,A 0.000,B 0.000,C 90.000,E1 274.588} C_DIS
LIN {X 0.130,Y -343.812,Z 1671.523,A 0.000,B 0.000,C 90.000,E1 274.188} C_DIS
LIN {X 0.150,Y -334.219,Z 1671.521,A 0.000,B 0.000,C 90.000,E1 273.669} C_DIS
LIN {X 0.052,Y -324.395,Z 1671.518,A 0.000,B 0.000,C 90.000,E1 273.212} C_DIS
LIN {X -0.045,Y -314.586,Z 1671.516,A 0.000,B 0.000,C 90.000,E1 272.808} C_DIS
LIN {X 0.069,Y -304.462,Z 1671.513,A 0.000,B 0.000,C 90.000,E1 272.407} C_DIS
LIN {X 0.061,Y -297.086,Z 1671.512,A 0.000,B 0.000,C 90.000,E1 272.178} C_DIS
LIN {X -0.028,Y -289.642,Z 1671.511,A 0.000,B 0.000,C 90.000,E1 272.007} C_DIS
LIN {X 0.034,Y -281.677,Z 1671.510,A 0.000,B 0.000,C 90.000,E1 271.835} C_DIS
LIN {X -0.049,Y -272.640,Z 1671.510,A 0.000,B 0.000,C 90.000,E1 271.718} C_DIS
LIN {X 0.093,Y -263.707,Z 1671.509,A 0.000,B 0.000,C 90.000,E1 271.604} C_DIS
LIN {X 0.106,Y -232.841,Z 1671.508,A 0.000,B 0.000,C 90.000,E1 271.489} C_DIS
LIN {X -0.028,Y -194.998,Z 1671.508,A 0.000,B 0.000,C 90.000,E1 271.375} C_DIS
LIN {X -0.033,Y -182.670,Z 1671.507,A 0.000,B 0.000,C 90.000,E1 271.318} C_DIS
LIN {X -0.052,Y -181.391,Z 1671.507,A 0.000,B 0.000,C 90.000,E1 271.318} C_DIS
LIN {X 0.001,Y -181.581,Z 1671.502,A 0.000,B 0.000,C 90.000,E1 270.286} C_DIS
LIN {X 0.006,Y -180.876,Z 1671.473,A 0.000,B 0.000,C 90.000,E1 265.065} C_DIS
LIN {X 0.062,Y -178.993,Z 1671.444,A 0.000,B 0.000,C 90.000,E1 259.982} C_DIS
LIN {X -0.020,Y -178.574,Z 1671.440,A 0.000,B 0.000,C 90.000,E1 259.162} C_DIS
LIN {X 0.042,Y -175.627,Z 1671.411,A 0.000,B 0.000,C 90.000,E1 254.047} C_DIS
LIN {X 0.103,Y -172.347,Z 1671.388,A 0.000,B 0.000,C 90.000,E1 249.752} C_DIS
LIN {X 0.055,Y -171.127,Z 1671.378,A 0.000,B 0.000,C 90.000,E1 248.050} C_DIS
LIN {X -0.058,Y -167.436,Z 1671.354,A 0.000,B 0.000,C 90.000,E1 243.768} C_DIS
LIN {X 0.023,Y -166.831,Z 1671.349,A 0.000,B 0.000,C 90.000,E1 242.871} C_DIS
LIN {X -0.059,Y -162.814,Z 1671.325,A 0.000,B 0.000,C 90.000,E1 238.535} C_DIS
LIN {X 0.004,Y -161.501,Z 1671.315,A 0.000,B 0.000,C 90.000,E1 236.755} C_DIS
LIN {X -0.042,Y -157.498,Z 1671.291,A 0.000,B 0.000,C 90.000,E1 232.351} C_DIS
LIN {X -0.008,Y -155.517,Z 1671.276,A 0.000,B 0.000,C 90.000,E1 229.666} C_DIS
LIN {X 0.042,Y -151.817,Z 1671.251,A 0.000,B 0.000,C 90.000,E1 225.162} C_DIS
LIN {X 0.054,Y -150.030,Z 1671.236,A 0.000,B 0.000,C 90.000,E1 222.447} C_DIS
LIN {X -0.031,Y -146.849,Z 1671.211,A 0.000,B 0.000,C 90.000,E1 217.935} C_DIS
LIN {X -0.014,Y -145.433,Z 1671.195,A 0.000,B 0.000,C 90.000,E1 215.185} C_DIS
LIN {X -0.017,Y -142.856,Z 1671.170,A 0.000,B 0.000,C 90.000,E1 210.590} C_DIS
LIN {X 0.035,Y -141.472,Z 1671.149,A 0.000,B 0.000,C 90.000,E1 206.873} C_DIS
LIN {X 0.026,Y -139.378,Z 1671.113,A 0.000,B 0.000,C 90.000,E1 200.375} C_DIS
LIN {X 0.015,Y -138.831,Z 1671.098,A 0.000,B 0.000,C 90.000,E1 197.583} C_DIS
LIN {X -0.056,Y -138.353,Z 1671.056,A 0.000,B 0.000,C 90.000,E1 190.141} C_DIS
LIN {X -0.061,Y -139.527,Z 1671.004,A 0.000,B 0.000,C 90.000,E1 180.802} C_DIS
LIN {X 0.031,Y -141.199,Z 1670.973,A 0.000,B 0.000,C 90.000,E1 175.179} C_DIS
LIN {X -0.009,Y -142.575,Z 1670.958,A 0.000,B 0.000,C 90.000,E1 172.413} C_DIS
LIN {X -0.055,Y -144.866,Z 1670.932,A 0.000,B 0.000,C 90.000,E1 167.813} C_DIS
LIN {X 0.041,Y -147.492,Z 1670.912,A 0.000,B 0.000,C 90.000,E1 164.102} C_DIS
LIN {X -0.025,Y -150.082,Z 1670.891,A 0.000,B 0.000,C 90.000,E1 160.477} C_DIS
LIN {X -0.011,Y -153.433,Z 1670.871,A 0.000,B 0.000,C 90.000,E1 156.847} C_DIS
LIN {X -0.024,Y -156.853,Z 1670.851,A 0.000,B 0.000,C 90.000,E1 153.256} C_DIS
LIN {X 0.047,Y -160.935,Z 1670.832,A 0.000,B 0.000,C 90.000,E1 149.665} C_DIS
LIN {X -0.009,Y -163.058,Z 1670.822,A 0.000,B 0.000,C 90.000,E1 147.916} C_DIS
LIN {X -0.005,Y -167.454,Z 1670.802,A 0.000,B 0.000,C 90.000,E1 144.402} C_DIS
LIN {X 0.039,Y -171.291,Z 1670.788,A 0.000,B 0.000,C 90.000,E1 141.778} C_DIS
LIN {X 0.074,Y -176.186,Z 1670.769,A 0.000,B 0.000,C 90.000,E1 138.324} C_DIS
LIN {X -0.060,Y -180.460,Z 1670.754,A 0.000,B 0.000,C 90.000,E1 135.810} C_DIS
LIN {X -0.086,Y -185.865,Z 1670.736,A 0.000,B 0.000,C 90.000,E1 132.447} C_DIS
LIN {X -0.033,Y -190.489,Z 1670.722,A 0.000,B 0.000,C 90.000,E1 129.930} C_DIS
LIN {X -0.011,Y -196.240,Z 1670.703,A 0.000,B 0.000,C 90.000,E1 126.629} C_DIS
LIN {X -0.054,Y -201.047,Z 1670.690,A 0.000,B 0.000,C 90.000,E1 124.199} C_DIS
LIN {X -0.041,Y -207.335,Z 1670.671,A 0.000,B 0.000,C 90.000,E1 120.797} C_DIS
LIN {X -0.059,Y -207.765,Z 1670.670,A 0.000,B 0.000,C 90.000,E1 120.590} C_DIS
LIN {X 0.130,Y -329.507,Z 1670.670,A 0.000,B 0.000,C 90.000,E1 120.541} C_DIS
LIN {X -0.048,Y -331.397,Z 1670.670,A 0.000,B 0.000,C 90.000,E1 120.541} C_DIS
LIN {X 0.090,Y -335.606,Z 1670.669,A 0.000,B 0.000,C 90.000,E1 120.335} C_DIS
LIN {X -0.063,Y -338.015,Z 1670.668,A 0.000,B 0.000,C 90.000,E1 120.178} C_DIS
LIN {X -0.123,Y -341.852,Z 1670.665,A 0.000,B 0.000,C 90.000,E1 119.745} C_DIS
LIN {X 0.052,Y -343.682,Z 1670.663,A 0.000,B 0.000,C 90.000,E1 119.411} C_DIS
LIN {X 0.030,Y -360.576,Z 1670.643,A 0.000,B 0.000,C 90.000,E1 115.771} C_DIS
LIN {X 0.194,Y -374.911,Z 1670.628,A 0.000,B 0.000,C 90.000,E1 113.078} C_DIS
LIN {X -0.012,Y -389.025,Z 1670.615,A 0.000,B 0.000,C 90.000,E1 110.791} C_DIS
LIN {X -0.154,Y -404.532,Z 1670.603,A 0.000,B 0.000,C 90.000,E1 108.544} C_DIS
LIN {X -0.046,Y -421.539,Z 1670.591,A 0.000,B 0.000,C 90.000,E1 106.315} C_DIS
LIN {X -0.173,Y -440.164,Z 1670.579,A 0.000,B 0.000,C 90.000,E1 104.175} C_DIS
LIN {X -0.119,Y -460.035,Z 1670.567,A 0.000,B 0.000,C 90.000,E1 102.119} C_DIS
LIN {X -0.171,Y -483.042,Z 1670.556,A 0.000,B 0.000,C 90.000,E1 100.018} C_DIS
LIN {X -0.199,Y -501.366,Z 1670.547,A 0.000,B 0.000,C 90.000,E1 98.511} C_DIS
LIN {X 0.178,Y -505.135,Z 1670.545,A 0.000,B 0.000,C 90.000,E1 98.049} C_DIS
LIN {X 0.110,Y -506.580,Z 1670.543,A 0.000,B 0.000,C 90.000,E1 97.814} C_DIS
LIN {X -0.027,Y -507.648,Z 1670.542,A 0.000,B 0.000,C 90.000,E1 97.587} C_DIS
LIN {X -0.204,Y -508.864,Z 1670.539,A 0.000,B 0.000,C 90.000,E1 97.125} C_DIS
LIN {X 0.130,Y -509.036,Z 1670.537,A 0.000,B 0.000,C 90.000,E1 96.606} C_DIS
LIN {X -0.034,Y -508.189,Z 1670.534,A 0.000,B 0.000,C 90.000,E1 96.144} C_DIS
LIN {X -0.198,Y -506.176,Z 1670.531,A 0.000,B 0.000,C 90.000,E1 95.682} C_DIS
LIN {X 0.135,Y -502.834,Z 1670.529,A 0.000,B 0.000,C 90.000,E1 95.163} C_DIS
LIN {X -0.176,Y -490.617,Z 1670.519,A 0.000,B 0.000,C 90.000,E1 93.498} C_DIS
LIN {X -0.083,Y -479.932,Z 1670.511,A 0.000,B 0.000,C 90.000,E1 92.007} C_DIS
LIN {X 0.106,Y -467.312,Z 1670.501,A 0.000,B 0.000,C 90.000,E1 90.229} C_DIS
LIN {X 0.023,Y -454.655,Z 1670.491,A 0.000,B 0.000,C 90.000,E1 88.453} C_DIS
LIN {X 0.210,Y -445.360,Z 1670.484,A 0.000,B 0.000,C 90.000,E1 87.135} C_DIS
LIN {X 0.157,Y -431.909,Z 1670.474,A 0.000,B 0.000,C 90.000,E1 85.298} C_DIS
LIN {X -0.073,Y -418.523,Z 1670.464,A 0.000,B 0.000,C 90.000,E1 83.451} C_DIS
LIN {X -0.004,Y -401.838,Z 1670.450,A 0.000,B 0.000,C 90.000,E1 80.971} C_DIS
LIN {X -0.184,Y -386.055,Z 1670.436,A 0.000,B 0.000,C 90.000,E1 78.465} C_DIS
LIN {X 0.116,Y -370.902,Z 1670.421,A 0.000,B 0.000,C 90.000,E1 75.825} C_DIS
LIN {X -0.066,Y -356.289,Z 1670.407,A 0.000,B 0.000,C 90.000,E1 73.196} C_DIS
LIN {X -0.167,Y -339.395,Z 1670.388,A 0.000,B 0.000,C 90.000,E1 69.880} C_DIS
LIN {X 0.059,Y -327.919,Z 1670.374,A 0.000,B 0.000,C 90.000,E1 67.358} C_DIS
LIN {X -0.046,Y -316.879,Z 1670.360,A 0.000,B 0.000,C 90.000,E1 64.845} C_DIS
LIN {X 0.131,Y -306.053,Z 1670.346,A 0.000,B 0.000,C 90.000,E1 62.231} C_DIS
LIN {X 0.017,Y -297.940,Z 1670.335,A 0.000,B 0.000,C 90.000,E1 60.284} C_DIS
LIN {X 0.054,Y -291.033,Z 1670.326,A 0.000,B 0.000,C 90.000,E1 58.614} C_DIS
LIN {X -0.130,Y -282.471,Z 1670.314,A 0.000,B 0.000,C 90.000,E1 56.628} C_DIS
LIN {X 0.017,Y -272.293,Z 1670.301,A 0.000,B 0.000,C 90.000,E1 54.196} C_DIS
LIN {X 0.040,Y -262.252,Z 1670.287,A 0.000,B 0.000,C 90.000,E1 51.743} C_DIS
LIN {X 0.026,Y -250.013,Z 1670.270,A 0.000,B 0.000,C 90.000,E1 48.528} C_DIS
LIN {X -0.011,Y -238.722,Z 1670.251,A 0.000,B 0.000,C 90.000,E1 45.243} C_DIS
LIN {X 0.030,Y -229.506,Z 1670.235,A 0.000,B 0.000,C 90.000,E1 42.243} C_DIS
LIN {X 0.047,Y -221.027,Z 1670.218,A 0.000,B 0.000,C 90.000,E1 39.197} C_DIS
LIN {X 0.092,Y -213.217,Z 1670.201,A 0.000,B 0.000,C 90.000,E1 36.091} C_DIS
LIN {X -0.125,Y -204.333,Z 1670.179,A 0.000,B 0.000,C 90.000,E1 32.212} C_DIS
LIN {X 0.078,Y -197.789,Z 1670.161,A 0.000,B 0.000,C 90.000,E1 28.949} C_DIS
LIN {X 0.003,Y -191.828,Z 1670.143,A 0.000,B 0.000,C 90.000,E1 25.720} C_DIS
LIN {X 0.059,Y -186.491,Z 1670.125,A 0.000,B 0.000,C 90.000,E1 22.408} C_DIS
LIN {X 0.016,Y -181.759,Z 1670.106,A 0.000,B 0.000,C 90.000,E1 19.087} C_DIS
LIN {X 0.018,Y -177.686,Z 1670.087,A 0.000,B 0.000,C 90.000,E1 15.717} C_DIS
LIN {X -0.030,Y -173.650,Z 1670.064,A 0.000,B 0.000,C 90.000,E1 11.478} C_DIS
LIN {X -0.018,Y -170.649,Z 1670.040,A 0.000,B 0.000,C 90.000,E1 7.182} C_DIS
LIN {X -0.076,Y -167.878,Z 1670.006,A 0.000,B 0.000,C 90.000,E1 1.146} C_DIS
LIN {X -0.077,Y -167.194,Z 1669.954,A 0.000,B 0.000,C 90.000,E1 351.724} C_DIS
LIN {X 0.066,Y -169.088,Z 1669.920,A 0.000,B 0.000,C 90.000,E1 345.589} C_DIS
LIN {X 0.025,Y -171.697,Z 1669.896,A 0.000,B 0.000,C 90.000,E1 341.275} C_DIS
LIN {X 0.031,Y -175.464,Z 1669.872,A 0.000,B 0.000,C 90.000,E1 336.975} C_DIS
LIN {X -0.046,Y -179.500,Z 1669.853,A 0.000,B 0.000,C 90.000,E1 333.589} C_DIS
LIN {X -0.031,Y -184.198,Z 1669.834,A 0.000,B 0.000,C 90.000,E1 330.205} C_DIS
LIN {X 0.066,Y -189.845,Z 1669.816,A 0.000,B 0.000,C 90.000,E1 326.834} C_DIS
LIN {X 0.047,Y -196.546,Z 1669.797,A 0.000,B 0.000,C 90.000,E1 323.543} C_DIS
LIN {X -0.034,Y -203.364,Z 1669.782,A 0.000,B 0.000,C 90.000,E1 320.723} C_DIS
LIN {X -0.114,Y -212.231,Z 1669.764,A 0.000,B 0.000,C 90.000,E1 317.553} C_DIS
LIN {X 0.028,Y -219.726,Z 1669.751,A 0.000,B 0.000,C 90.000,E1 315.162} C_DIS
LIN {X 0.099,Y -229.453,Z 1669.736,A 0.000,B 0.000,C 90.000,E1 312.447} C_DIS
LIN {X -0.079,Y -240.245,Z 1669.721,A 0.000,B 0.000,C 90.000,E1 309.850} C_DIS
LIN {X 0.036,Y -248.808,Z 1669.711,A 0.000,B 0.000,C 90.000,E1 307.971} C_DIS
LIN {X 0.018,Y -262.282,Z 1669.697,A 0.000,B 0.000,C 90.000,E1 305.438} C_DIS
LIN {X 0.056,Y -277.046,Z 1669.683,A 0.000,B 0.000,C 90.000,E1 302.959} C_DIS
LIN {X -0.123,Y -295.599,Z 1669.668,A 0.000,B 0.000,C 90.000,E1 300.256} C_DIS
LIN {X -0.015,Y -315.356,Z 1669.653,A 0.000,B 0.000,C 90.000,E1 297.590} C_DIS
LIN {X 0.037,Y -327.900,Z 1669.644,A 0.000,B 0.000,C 90.000,E1 295.976} C_DIS
LIN {X 0.126,Y -342.659,Z 1669.634,A 0.000,B 0.000,C 90.000,E1 294.079} C_DIS
LIN {X -0.100,Y -357.557,Z 1669.624,A 0.000,B 0.000,C 90.000,E1 292.280} C_DIS
LIN {X -0.147,Y -369.703,Z 1669.615,A 0.000,B 0.000,C 90.000,E1 290.791} C_DIS
LIN {X 0.000,Y -376.597,Z 1669.610,A 0.000,B 0.000,C 90.000,E1 289.885} C_DIS
LIN {X -0.147,Y -382.998,Z 1669.606,A 0.000,B 0.000,C 90.000,E1 289.033} C_DIS
LIN {X 0.113,Y -386.991,Z 1669.602,A 0.000,B 0.000,C 90.000,E1 288.417} C_DIS
LIN {X -0.056,Y -392.280,Z 1669.598,A 0.000,B 0.000,C 90.000,E1 287.583} C_DIS
LIN {X 0.147,Y -395.315,Z 1669.594,A 0.000,B 0.000,C 90.000,E1 286.985} C_DIS
LIN {X 0.054,Y -399.104,Z 1669.590,A 0.000,B 0.000,C 90.000,E1 286.150} C_DIS
LIN {X -0.079,Y -401.188,Z 1669.587,A 0.000,B 0.000,C 90.000,E1 285.607} C_DIS
LIN {X 0.185,Y -402.864,Z 1669.583,A 0.000,B 0.000,C 90.000,E1 285.009} C_DIS
LIN {X -0.038,Y -404.258,Z 1669.580,A 0.000,B 0.000,C 90.000,E1 284.481} C_DIS
LIN {X -0.151,Y -405.157,Z 1669.577,A 0.000,B 0.000,C 90.000,E1 283.939} C_DIS
LIN {X 0.038,Y -405.713,Z 1669.574,A 0.000,B 0.000,C 90.000,E1 283.355} C_DIS
LIN {X -0.160,Y -405.779,Z 1669.571,A 0.000,B 0.000,C 90.000,E1 282.827} C_DIS
LIN {X 0.042,Y -405.426,Z 1669.568,A 0.000,B 0.000,C 90.000,E1 282.243} C_DIS
LIN {X -0.151,Y -404.560,Z 1669.565,A 0.000,B 0.000,C 90.000,E1 281.715} C_DIS
LIN {X 0.050,Y -403.235,Z 1669.562,A 0.000,B 0.000,C 90.000,E1 281.130} C_DIS
LIN {X -0.151,Y -401.329,Z 1669.559,A 0.000,B 0.000,C 90.000,E1 280.602} C_DIS
LIN {X 0.033,Y -398.849,Z 1669.556,A 0.000,B 0.000,C 90.000,E1 280.018} C_DIS
LIN {X -0.186,Y -394.045,Z 1669.551,A 0.000,B 0.000,C 90.000,E1 279.208} C_DIS
LIN {X -0.048,Y -388.373,Z 1669.546,A 0.000,B 0.000,C 90.000,E1 278.341} C_DIS
LIN {X 0.035,Y -381.961,Z 1669.542,A 0.000,B 0.000,C 90.000,E1 277.473} C_DIS
LIN {X 0.089,Y -377.095,Z 1669.538,A 0.000,B 0.000,C 90.000,E1 276.891} C_DIS
LIN {X 0.112,Y -371.735,Z 1669.535,A 0.000,B 0.000,C 90.000,E1 276.315} C_DIS
LIN {X -0.083,Y -365.884,Z 1669.532,A 0.000,B 0.000,C 90.000,E1 275.796} C_DIS
LIN {X -0.010,Y -359.757,Z 1669.529,A 0.000,B 0.000,C 90.000,E1 275.277} C_DIS
LIN {X -0.038,Y -353.356,Z 1669.527,A 0.000,B 0.000,C 90.000,E1 274.821} C_DIS
LIN {X -0.080,Y -346.763,Z 1669.524,A 0.000,B 0.000,C 90.000,E1 274.416} C_DIS
LIN {X 0.129,Y -337.003,Z 1669.521,A 0.000,B 0.000,C 90.000,E1 273.841} C_DIS
LIN {X -0.007,Y -327.389,Z 1669.519,A 0.000,B 0.000,C 90.000,E1 273.383} C_DIS
LIN {X 0.107,Y -317.470,Z 1669.516,A 0.000,B 0.000,C 90.000,E1 272.922} C_DIS
LIN {X -0.144,Y -307.545,Z 1669.514,A 0.000,B 0.000,C 90.000,E1 272.579} C_DIS
LIN {X 0.119,Y -300.696,Z 1669.513,A 0.000,B 0.000,C 90.000,E1 272.293} C_DIS
LIN {X -0.066,Y -293.261,Z 1669.512,A 0.000,B 0.000,C 90.000,E1 272.121} C_DIS
LIN {X -0.065,Y -285.611,Z 1669.511,A 0.000,B 0.000,C 90.000,E1 271.949} C_DIS
LIN {X 0.081,Y -276.971,Z 1669.510,A 0.000,B 0.000,C 90.000,E1 271.776} C_DIS
LIN {X 0.053,Y -266.225,Z 1669.509,A 0.000,B 0.000,C 90.000,E1 271.661} C_DIS
LIN {X 0.055,Y -241.046,Z 1669.509,A 0.000,B 0.000,C 90.000,E1 271.547} C_DIS
LIN {X 0.032,Y -196.024,Z 1669.508,A 0.000,B 0.000,C 90.000,E1 271.375} C_DIS
LIN {X 0.013,Y -183.348,Z 1669.507,A 0.000,B 0.000,C 90.000,E1 271.318} C_DIS
LIN {X -0.007,Y -181.388,Z 1669.507,A 0.000,B 0.000,C 90.000,E1 271.318} C_DIS
LIN {X -0.052,Y -181.572,Z 1669.502,A 0.000,B 0.000,C 90.000,E1 270.458} C_DIS
LIN {X -0.074,Y -180.906,Z 1669.474,A 0.000,B 0.000,C 90.000,E1 265.412} C_DIS
LIN {X 0.000,Y -180.699,Z 1669.470,A 0.000,B 0.000,C 90.000,E1 264.546} C_DIS
LIN {X 0.077,Y -178.784,Z 1669.442,A 0.000,B 0.000,C 90.000,E1 259.454} C_DIS
LIN {X -0.020,Y -175.829,Z 1669.413,A 0.000,B 0.000,C 90.000,E1 254.393} C_DIS
LIN {X -0.020,Y -172.018,Z 1669.385,A 0.000,B 0.000,C 90.000,E1 249.263} C_DIS
LIN {X -0.044,Y -171.442,Z 1669.380,A 0.000,B 0.000,C 90.000,E1 248.411} C_DIS
LIN {X 0.011,Y -167.677,Z 1669.356,A 0.000,B 0.000,C 90.000,E1 244.076} C_DIS
LIN {X -0.048,Y -166.352,Z 1669.346,A 0.000,B 0.000,C 90.000,E1 242.359} C_DIS
LIN {X -0.056,Y -163.086,Z 1669.327,A 0.000,B 0.000,C 90.000,E1 238.869} C_DIS
LIN {X -0.005,Y -161.029,Z 1669.312,A 0.000,B 0.000,C 90.000,E1 236.215} C_DIS
LIN {X -0.021,Y -157.769,Z 1669.293,A 0.000,B 0.000,C 90.000,E1 232.683} C_DIS
LIN {X 0.042,Y -155.807,Z 1669.278,A 0.000,B 0.000,C 90.000,E1 229.989} C_DIS
LIN {X -0.010,Y -152.059,Z 1669.253,A 0.000,B 0.000,C 90.000,E1 225.526} C_DIS
LIN {X 0.003,Y -150.309,Z 1669.238,A 0.000,B 0.000,C 90.000,E1 222.813} C_DIS
LIN {X 0.039,Y -147.053,Z 1669.213,A 0.000,B 0.000,C 90.000,E1 218.257} C_DIS
LIN {X 0.031,Y -145.631,Z 1669.197,A 0.000,B 0.000,C 90.000,E1 215.518} C_DIS
LIN {X 0.029,Y -143.014,Z 1669.172,A 0.000,B 0.000,C 90.000,E1 210.924} C_DIS
LIN {X -0.040,Y -141.640,Z 1669.151,A 0.000,B 0.000,C 90.000,E1 207.257} C_DIS
LIN {X 0.011,Y -139.439,Z 1669.115,A 0.000,B 0.000,C 90.000,E1 200.737} C_DIS
LIN {X -0.068,Y -139.171,Z 1669.105,A 0.000,B 0.000,C 90.000,E1 198.906} C_DIS
LIN {X -0.039,Y -138.318,Z 1669.053,A 0.000,B 0.000,C 90.000,E1 189.557} C_DIS
LIN {X -0.030,Y -139.472,Z 1669.006,A 0.000,B 0.000,C 90.000,E1 181.146} C_DIS
LIN {X 0.051,Y -141.047,Z 1668.975,A 0.000,B 0.000,C 90.000,E1 175.527} C_DIS
LIN {X 0.005,Y -142.416,Z 1668.960,A 0.000,B 0.000,C 90.000,E1 172.761} C_DIS
LIN {X -0.075,Y -144.651,Z 1668.934,A 0.000,B 0.000,C 90.000,E1 168.173} C_DIS
LIN {X -0.016,Y -147.848,Z 1668.909,A 0.000,B 0.000,C 90.000,E1 163.559} C_DIS
LIN {X 0.069,Y -150.548,Z 1668.888,A 0.000,B 0.000,C 90.000,E1 159.880} C_DIS
LIN {X -0.053,Y -154.014,Z 1668.868,A 0.000,B 0.000,C 90.000,E1 156.305} C_DIS
LIN {X 0.006,Y -157.429,Z 1668.848,A 0.000,B 0.000,C 90.000,E1 152.692} C_DIS
LIN {X 0.028,Y -161.642,Z 1668.828,A 0.000,B 0.000,C 90.000,E1 149.125} C_DIS
LIN {X 0.046,Y -165.837,Z 1668.809,A 0.000,B 0.000,C 90.000,E1 145.595} C_DIS
LIN {X 0.038,Y -170.809,Z 1668.790,A 0.000,B 0.000,C 90.000,E1 142.110} C_DIS
LIN {X -0.046,Y -175.679,Z 1668.770,A 0.000,B 0.000,C 90.000,E1 138.690} C_DIS
LIN {X 0.079,Y -181.292,Z 1668.751,A 0.000,B 0.000,C 90.000,E1 135.243} C_DIS
LIN {X -0.049,Y -186.772,Z 1668.733,A 0.000,B 0.000,C 90.000,E1 131.919} C_DIS
LIN {X 0.022,Y -191.365,Z 1668.719,A 0.000,B 0.000,C 90.000,E1 129.402} C_DIS
LIN {X 0.105,Y -197.205,Z 1668.701,A 0.000,B 0.000,C 90.000,E1 126.091} C_DIS
LIN {X 0.029,Y -200.483,Z 1668.692,A 0.000,B 0.000,C 90.000,E1 124.485} C_DIS
LIN {X 0.030,Y -207.655,Z 1668.670,A 0.000,B 0.000,C 90.000,E1 120.620} C_DIS
LIN {X 0.069,Y -207.693,Z 1668.670,A 0.000,B 0.000,C 90.000,E1 120.590} C_DIS
LIN {X 0.075,Y -329.123,Z 1668.670,A 0.000,B 0.000,C 90.000,E1 120.590} C_DIS
LIN {X 0.055,Y -333.925,Z 1668.669,A 0.000,B 0.000,C 90.000,E1 120.463} C_DIS
LIN {X -0.213,Y -336.709,Z 1668.668,A 0.000,B 0.000,C 90.000,E1 120.335} C_DIS
LIN {X 0.009,Y -340.477,Z 1668.666,A 0.000,B 0.000,C 90.000,E1 119.922} C_DIS
LIN {X -0.213,Y -343.916,Z 1668.663,A 0.000,B 0.000,C 90.000,E1 119.411} C_DIS
LIN {X -0.198,Y -357.815,Z 1668.646,A 0.000,B 0.000,C 90.000,E1 116.360} C_DIS
LIN {X 0.041,Y -371.825,Z 1668.631,A 0.000,B 0.000,C 90.000,E1 113.643} C_DIS
LIN {X -0.103,Y -385.633,Z 1668.618,A 0.000,B 0.000,C 90.000,E1 111.334} C_DIS
LIN {X 0.041,Y -400.809,Z 1668.606,A 0.000,B 0.000,C 90.000,E1 109.033} C_DIS
LIN {X 0.071,Y -417.460,Z 1668.593,A 0.000,B 0.000,C 90.000,E1 106.804} C_DIS
LIN {X -0.027,Y -435.701,Z 1668.581,A 0.000,B 0.000,C 90.000,E1 104.647} C_DIS
LIN {X 0.206,Y -455.373,Z 1668.570,A 0.000,B 0.000,C 90.000,E1 102.535} C_DIS
LIN {X -0.143,Y -475.681,Z 1668.559,A 0.000,B 0.000,C 90.000,E1 100.658} C_DIS
LIN {X 0.012,Y -501.688,Z 1668.547,A 0.000,B 0.000,C 90.000,E1 98.454} C_DIS
LIN {X 0.253,Y -503.679,Z 1668.546,A 0.000,B 0.000,C 90.000,E1 98.219} C_DIS
LIN {X 0.117,Y -505.438,Z 1668.544,A 0.000,B 0.000,C 90.000,E1 97.992} C_DIS
LIN {X 0.049,Y -506.753,Z 1668.543,A 0.000,B 0.000,C 90.000,E1 97.757} C_DIS
LIN {X -0.136,Y -508.370,Z 1668.540,A 0.000,B 0.000,C 90.000,E1 97.296} C_DIS
LIN {X 0.191,Y -508.891,Z 1668.538,A 0.000,B 0.000,C 90.000,E1 96.777} C_DIS
LIN {X 0.023,Y -508.402,Z 1668.535,A 0.000,B 0.000,C 90.000,E1 96.315} C_DIS
LIN {X -0.143,Y -506.823,Z 1668.532,A 0.000,B 0.000,C 90.000,E1 95.853} C_DIS
LIN {X -0.252,Y -505.535,Z 1668.531,A 0.000,B 0.000,C 90.000,E1 95.625} C_DIS
LIN {X 0.031,Y -493.369,Z 1668.522,A 0.000,B 0.000,C 90.000,E1 93.898} C_DIS
LIN {X 0.161,Y -482.786,Z 1668.513,A 0.000,B 0.000,C 90.000,E1 92.407} C_DIS
LIN {X -0.075,Y -470.203,Z 1668.504,A 0.000,B 0.000,C 90.000,E1 90.688} C_DIS
LIN {X -0.090,Y -457.573,Z 1668.494,A 0.000,B 0.000,C 90.000,E1 88.912} C_DIS
LIN {X -0.101,Y -446.513,Z 1668.485,A 0.000,B 0.000,C 90.000,E1 87.364} C_DIS
LIN {X -0.118,Y -433.051,Z 1668.475,A 0.000,B 0.000,C 90.000,E1 85.527} C_DIS
LIN {X 0.057,Y -419.626,Z 1668.465,A 0.000,B 0.000,C 90.000,E1 83.628} C_DIS
LIN {X -0.094,Y -401.031,Z 1668.449,A 0.000,B 0.000,C 90.000,E1 80.905} C_DIS
LIN {X 0.095,Y -385.275,Z 1668.435,A 0.000,B 0.000,C 90.000,E1 78.342} C_DIS
LIN {X 0.019,Y -370.144,Z 1668.421,A 0.000,B 0.000,C 90.000,E1 75.755} C_DIS
LIN {X 0.064,Y -355.528,Z 1668.406,A 0.000,B 0.000,C 90.000,E1 73.087} C_DIS
LIN {X 0.042,Y -338.701,Z 1668.388,A 0.000,B 0.000,C 90.000,E1 69.752} C_DIS
LIN {X -0.056,Y -327.228,Z 1668.374,A 0.000,B 0.000,C 90.000,E1 67.283} C_DIS
LIN {X 0.119,Y -316.190,Z 1668.360,A 0.000,B 0.000,C 90.000,E1 64.717} C_DIS
LIN {X 0.004,Y -305.379,Z 1668.345,A 0.000,B 0.000,C 90.000,E1 62.153} C_DIS
LIN {X -0.116,Y -297.255,Z 1668.334,A 0.000,B 0.000,C 90.000,E1 60.205} C_DIS
LIN {X -0.086,Y -290.315,Z 1668.325,A 0.000,B 0.000,C 90.000,E1 58.535} C_DIS
LIN {X -0.041,Y -281.740,Z 1668.314,A 0.000,B 0.000,C 90.000,E1 56.501} C_DIS
LIN {X -0.044,Y -270.102,Z 1668.299,A 0.000,B 0.000,C 90.000,E1 53.749} C_DIS
LIN {X 0.043,Y -257.393,Z 1668.281,A 0.000,B 0.000,C 90.000,E1 50.561} C_DIS
LIN {X 0.056,Y -245.508,Z 1668.263,A 0.000,B 0.000,C 90.000,E1 47.310} C_DIS
LIN {X -0.111,Y -234.666,Z 1668.245,A 0.000,B 0.000,C 90.000,E1 44.028} C_DIS
LIN {X -0.003,Y -225.767,Z 1668.228,A 0.000,B 0.000,C 90.000,E1 40.987} C_DIS
LIN {X -0.048,Y -217.571,Z 1668.211,A 0.000,B 0.000,C 90.000,E1 37.935} C_DIS
LIN {X -0.043,Y -210.032,Z 1668.193,A 0.000,B 0.000,C 90.000,E1 34.818} C_DIS
LIN {X -0.110,Y -203.059,Z 1668.176,A 0.000,B 0.000,C 90.000,E1 31.671} C_DIS
LIN {X -0.036,Y -196.621,Z 1668.158,A 0.000,B 0.000,C 90.000,E1 28.437} C_DIS
LIN {X 0.038,Y -190.740,Z 1668.140,A 0.000,B 0.000,C 90.000,E1 25.155} C_DIS
LIN {X 0.066,Y -185.552,Z 1668.121,A 0.000,B 0.000,C 90.000,E1 21.844} C_DIS
LIN {X -0.063,Y -180.941,Z 1668.103,A 0.000,B 0.000,C 90.000,E1 18.544} C_DIS
LIN {X 0.043,Y -177.031,Z 1668.084,A 0.000,B 0.000,C 90.000,E1 15.134} C_DIS
LIN {X -0.019,Y -173.158,Z 1668.061,A 0.000,B 0.000,C 90.000,E1 10.894} C_DIS
LIN {X -0.035,Y -169.818,Z 1668.032,A 0.000,B 0.000,C 90.000,E1 5.739} C_DIS
LIN {X -0.030,Y -167.516,Z 1667.997,A 0.000,B 0.000,C 90.000,E1 359.542} C_DIS
LIN {X -0.014,Y -168.353,Z 1667.930,A 0.000,B 0.000,C 90.000,E1 347.353} C_DIS
LIN {X 0.064,Y -171.117,Z 1667.901,A 0.000,B 0.000,C 90.000,E1 342.127} C_DIS
LIN {X -0.015,Y -174.669,Z 1667.877,A 0.000,B 0.000,C 90.000,E1 337.847} C_DIS
LIN {X 0.053,Y -178.505,Z 1667.858,A 0.000,B 0.000,C 90.000,E1 334.409} C_DIS
LIN {X -0.038,Y -183.063,Z 1667.839,A 0.000,B 0.000,C 90.000,E1 331.051} C_DIS
LIN {X 0.094,Y -188.468,Z 1667.821,A 0.000,B 0.000,C 90.000,E1 327.661} C_DIS
LIN {X -0.073,Y -194.954,Z 1667.802,A 0.000,B 0.000,C 90.000,E1 324.402} C_DIS
LIN {X -0.038,Y -201.475,Z 1667.786,A 0.000,B 0.000,C 90.000,E1 321.537} C_DIS
LIN {X 0.100,Y -208.963,Z 1667.771,A 0.000,B 0.000,C 90.000,E1 318.690} C_DIS
LIN {X -0.059,Y -217.300,Z 1667.755,A 0.000,B 0.000,C 90.000,E1 315.972} C_DIS
LIN {X -0.047,Y -226.743,Z 1667.740,A 0.000,B 0.000,C 90.000,E1 313.257} C_DIS
LIN {X -0.129,Y -237.201,Z 1667.725,A 0.000,B 0.000,C 90.000,E1 310.620} C_DIS
LIN {X -0.102,Y -245.398,Z 1667.715,A 0.000,B 0.000,C 90.000,E1 308.749} C_DIS
LIN {X 0.108,Y -254.518,Z 1667.705,A 0.000,B 0.000,C 90.000,E1 306.870} C_DIS
LIN {X -0.033,Y -270.632,Z 1667.689,A 0.000,B 0.000,C 90.000,E1 304.040} C_DIS
LIN {X 0.044,Y -286.246,Z 1667.676,A 0.000,B 0.000,C 90.000,E1 301.592} C_DIS
LIN {X 0.062,Y -305.403,Z 1667.661,A 0.000,B 0.000,C 90.000,E1 298.899} C_DIS
LIN {X 0.090,Y -322.998,Z 1667.648,A 0.000,B 0.000,C 90.000,E1 296.616} C_DIS
LIN {X 0.113,Y -335.321,Z 1667.639,A 0.000,B 0.000,C 90.000,E1 295.027} C_DIS
LIN {X -0.110,Y -350.159,Z 1667.629,A 0.000,B 0.000,C 90.000,E1 293.206} C_DIS
LIN {X 0.074,Y -362.447,Z 1667.620,A 0.000,B 0.000,C 90.000,E1 291.663} C_DIS
LIN {X 0.019,Y -372.012,Z 1667.614,A 0.000,B 0.000,C 90.000,E1 290.482} C_DIS
LIN {X -0.172,Y -378.780,Z 1667.609,A 0.000,B 0.000,C 90.000,E1 289.631} C_DIS
LIN {X 0.066,Y -384.989,Z 1667.604,A 0.000,B 0.000,C 90.000,E1 288.725} C_DIS
LIN {X -0.009,Y -390.618,Z 1667.599,A 0.000,B 0.000,C 90.000,E1 287.873} C_DIS
LIN {X 0.182,Y -393.872,Z 1667.596,A 0.000,B 0.000,C 90.000,E1 287.275} C_DIS
LIN {X 0.077,Y -397.959,Z 1667.591,A 0.000,B 0.000,C 90.000,E1 286.441} C_DIS
LIN {X 0.006,Y -401.227,Z 1667.587,A 0.000,B 0.000,C 90.000,E1 285.607} C_DIS
LIN {X -0.118,Y -402.967,Z 1667.584,A 0.000,B 0.000,C 90.000,E1 285.064} C_DIS
LIN {X 0.049,Y -404.326,Z 1667.580,A 0.000,B 0.000,C 90.000,E1 284.481} C_DIS
LIN {X -0.064,Y -405.301,Z 1667.577,A 0.000,B 0.000,C 90.000,E1 283.939} C_DIS
LIN {X 0.125,Y -405.821,Z 1667.574,A 0.000,B 0.000,C 90.000,E1 283.355} C_DIS
LIN {X -0.072,Y -405.937,Z 1667.571,A 0.000,B 0.000,C 90.000,E1 282.827} C_DIS
LIN {X 0.131,Y -405.560,Z 1667.568,A 0.000,B 0.000,C 90.000,E1 282.243} C_DIS
LIN {X -0.061,Y -404.757,Z 1667.565,A 0.000,B 0.000,C 90.000,E1 281.715} C_DIS
LIN {X 0.140,Y -403.401,Z 1667.562,A 0.000,B 0.000,C 90.000,E1 281.130} C_DIS
LIN {X -0.060,Y -401.505,Z 1667.559,A 0.000,B 0.000,C 90.000,E1 280.602} C_DIS
LIN {X 0.125,Y -399.008,Z 1667.556,A 0.000,B 0.000,C 90.000,E1 280.018} C_DIS
LIN {X -0.169,Y -395.936,Z 1667.553,A 0.000,B 0.000,C 90.000,E1 279.500} C_DIS
LIN {X 0.040,Y -390.510,Z 1667.548,A 0.000,B 0.000,C 90.000,E1 278.624} C_DIS
LIN {X 0.142,Y -384.291,Z 1667.543,A 0.000,B 0.000,C 90.000,E1 277.757} C_DIS
LIN {X 0.161,Y -379.712,Z 1667.540,A 0.000,B 0.000,C 90.000,E1 277.182} C_DIS
LIN {X 0.156,Y -374.523,Z 1667.537,A 0.000,B 0.000,C 90.000,E1 276.606} C_DIS
LIN {X -0.119,Y -368.966,Z 1667.534,A 0.000,B 0.000,C 90.000,E1 276.087} C_DIS
LIN {X 0.167,Y -362.920,Z 1667.531,A 0.000,B 0.000,C 90.000,E1 275.511} C_DIS
LIN {X 0.001,Y -356.557,Z 1667.528,A 0.000,B 0.000,C 90.000,E1 275.049} C_DIS
LIN {X 0.174,Y -349.927,Z 1667.526,A 0.000,B 0.000,C 90.000,E1 274.588} C_DIS
LIN {X -0.056,Y -340.349,Z 1667.523,A 0.000,B 0.000,C 90.000,E1 274.073} C_DIS
LIN {X 0.046,Y -330.689,Z 1667.520,A 0.000,B 0.000,C 90.000,E1 273.555} C_DIS
LIN {X 0.085,Y -320.888,Z 1667.517,A 0.000,B 0.000,C 90.000,E1 273.094} C_DIS
LIN {X -0.008,Y -310.815,Z 1667.515,A 0.000,B 0.000,C 90.000,E1 272.694} C_DIS
LIN {X -0.075,Y -300.665,Z 1667.513,A 0.000,B 0.000,C 90.000,E1 272.350} C_DIS
LIN {X 0.052,Y -293.456,Z 1667.512,A 0.000,B 0.000,C 90.000,E1 272.121} C_DIS
LIN {X 0.060,Y -285.835,Z 1667.511,A 0.000,B 0.000,C 90.000,E1 271.949} C_DIS
LIN {X -0.073,Y -277.450,Z 1667.510,A 0.000,B 0.000,C 90.000,E1 271.835} C_DIS
LIN {X -0.073,Y -266.963,Z 1667.509,A 0.000,B 0.000,C 90.000,E1 271.718} C_DIS
LIN {X -0.024,Y -229.630,Z 1667.509,A 0.000,B 0.000,C 90.000,E1 271.547} C_DIS
LIN {X 0.048,Y -182.736,Z 1667.507,A 0.000,B 0.000,C 90.000,E1 271.318} C_DIS
LIN {X 0.028,Y -181.386,Z 1667.507,A 0.000,B 0.000,C 90.000,E1 271.318} C_DIS
LIN {X 0.005,Y -181.570,Z 1667.503,A 0.000,B 0.000,C 90.000,E1 270.458} C_DIS
LIN {X 0.046,Y -181.001,Z 1667.484,A 0.000,B 0.000,C 90.000,E1 267.078} C_DIS
LIN {X -0.018,Y -180.906,Z 1667.474,A 0.000,B 0.000,C 90.000,E1 265.412} C_DIS
LIN {X 0.039,Y -180.708,Z 1667.470,A 0.000,B 0.000,C 90.000,E1 264.552} C_DIS
LIN {X -0.042,Y -178.793,Z 1667.442,A 0.000,B 0.000,C 90.000,E1 259.511} C_DIS
LIN {X 0.036,Y -175.840,Z 1667.413,A 0.000,B 0.000,C 90.000,E1 254.393} C_DIS
LIN {X 0.036,Y -172.029,Z 1667.385,A 0.000,B 0.000,C 90.000,E1 249.263} C_DIS
LIN {X 0.012,Y -171.457,Z 1667.380,A 0.000,B 0.000,C 90.000,E1 248.411} C_DIS
LIN {X -0.008,Y -167.689,Z 1667.356,A 0.000,B 0.000,C 90.000,E1 244.101} C_DIS
LIN {X 0.006,Y -166.371,Z 1667.346,A 0.000,B 0.000,C 90.000,E1 242.359} C_DIS
LIN {X -0.003,Y -163.102,Z 1667.327,A 0.000,B 0.000,C 90.000,E1 238.869} C_DIS
LIN {X 0.048,Y -161.048,Z 1667.312,A 0.000,B 0.000,C 90.000,E1 236.215} C_DIS
LIN {X 0.031,Y -157.785,Z 1667.293,A 0.000,B 0.000,C 90.000,E1 232.683} C_DIS
LIN {X -0.026,Y -155.821,Z 1667.278,A 0.000,B 0.000,C 90.000,E1 230.033} C_DIS
LIN {X -0.068,Y -152.072,Z 1667.253,A 0.000,B 0.000,C 90.000,E1 225.567} C_DIS
LIN {X -0.049,Y -150.322,Z 1667.238,A 0.000,B 0.000,C 90.000,E1 222.852} C_DIS
LIN {X -0.027,Y -147.064,Z 1667.213,A 0.000,B 0.000,C 90.000,E1 218.302} C_DIS
LIN {X 0.081,Y -145.640,Z 1667.198,A 0.000,B 0.000,C 90.000,E1 215.518} C_DIS
LIN {X 0.077,Y -143.023,Z 1667.172,A 0.000,B 0.000,C 90.000,E1 210.924} C_DIS
LIN {X 0.009,Y -141.648,Z 1667.151,A 0.000,B 0.000,C 90.000,E1 207.257} C_DIS
LIN {X 0.059,Y -139.443,Z 1667.115,A 0.000,B 0.000,C 90.000,E1 200.737} C_DIS
LIN {X -0.020,Y -139.176,Z 1667.105,A 0.000,B 0.000,C 90.000,E1 198.906} C_DIS
LIN {X 0.009,Y -138.319,Z 1667.053,A 0.000,B 0.000,C 90.000,E1 189.557} C_DIS
LIN {X 0.018,Y -139.469,Z 1667.006,A 0.000,B 0.000,C 90.000,E1 181.146} C_DIS
LIN {X -0.041,Y -141.038,Z 1666.975,A 0.000,B 0.000,C 90.000,E1 175.584} C_DIS
LIN {X 0.054,Y -142.406,Z 1666.960,A 0.000,B 0.000,C 90.000,E1 172.761} C_DIS
LIN {X -0.025,Y -144.640,Z 1666.934,A 0.000,B 0.000,C 90.000,E1 168.173} C_DIS
LIN {X 0.035,Y -147.835,Z 1666.909,A 0.000,B 0.000,C 90.000,E1 163.559} C_DIS
LIN {X -0.021,Y -150.531,Z 1666.888,A 0.000,B 0.000,C 90.000,E1 159.934} C_DIS
LIN {X -0.002,Y -153.995,Z 1666.868,A 0.000,B 0.000,C 90.000,E1 156.305} C_DIS
LIN {X -0.081,Y -157.408,Z 1666.848,A 0.000,B 0.000,C 90.000,E1 152.743} C_DIS
LIN {X -0.002,Y -161.617,Z 1666.829,A 0.000,B 0.000,C 90.000,E1 149.154} C_DIS
LIN {X 0.100,Y -165.813,Z 1666.809,A 0.000,B 0.000,C 90.000,E1 145.595} C_DIS
LIN {X -0.012,Y -170.780,Z 1666.790,A 0.000,B 0.000,C 90.000,E1 142.145} C_DIS
LIN {X 0.010,Y -175.651,Z 1666.771,A 0.000,B 0.000,C 90.000,E1 138.690} C_DIS
LIN {X 0.008,Y -181.266,Z 1666.752,A 0.000,B 0.000,C 90.000,E1 135.283} C_DIS
LIN {X 0.008,Y -186.741,Z 1666.733,A 0.000,B 0.000,C 90.000,E1 131.919} C_DIS
LIN {X -0.040,Y -191.337,Z 1666.719,A 0.000,B 0.000,C 90.000,E1 129.439} C_DIS
LIN {X 0.006,Y -197.171,Z 1666.701,A 0.000,B 0.000,C 90.000,E1 126.137} C_DIS
LIN {X -0.075,Y -200.449,Z 1666.692,A 0.000,B 0.000,C 90.000,E1 124.532} C_DIS
LIN {X -0.061,Y -207.606,Z 1666.670,A 0.000,B 0.000,C 90.000,E1 120.669} C_DIS
LIN {X -0.133,Y -328.442,Z 1666.670,A 0.000,B 0.000,C 90.000,E1 120.669} C_DIS
LIN {X 0.155,Y -334.178,Z 1666.669,A 0.000,B 0.000,C 90.000,E1 120.463} C_DIS
LIN {X -0.111,Y -336.802,Z 1666.668,A 0.000,B 0.000,C 90.000,E1 120.335} C_DIS
LIN {X -0.004,Y -340.610,Z 1666.666,A 0.000,B 0.000,C 90.000,E1 119.922} C_DIS
LIN {X -0.165,Y -342.511,Z 1666.665,A 0.000,B 0.000,C 90.000,E1 119.667} C_DIS
LIN {X 0.144,Y -344.007,Z 1666.663,A 0.000,B 0.000,C 90.000,E1 119.333} C_DIS
LIN {X 0.020,Y -357.873,Z 1666.646,A 0.000,B 0.000,C 90.000,E1 116.309} C_DIS
LIN {X -0.064,Y -371.892,Z 1666.631,A 0.000,B 0.000,C 90.000,E1 113.643} C_DIS
LIN {X 0.150,Y -385.707,Z 1666.618,A 0.000,B 0.000,C 90.000,E1 111.280} C_DIS
LIN {X -0.069,Y -400.893,Z 1666.606,A 0.000,B 0.000,C 90.000,E1 109.033} C_DIS
LIN {X -0.040,Y -417.555,Z 1666.593,A 0.000,B 0.000,C 90.000,E1 106.804} C_DIS
LIN {X -0.142,Y -435.807,Z 1666.581,A 0.000,B 0.000,C 90.000,E1 104.647} C_DIS
LIN {X 0.094,Y -455.486,Z 1666.570,A 0.000,B 0.000,C 90.000,E1 102.535} C_DIS
LIN {X 0.215,Y -475.798,Z 1666.559,A 0.000,B 0.000,C 90.000,E1 100.602} C_DIS
LIN {X -0.093,Y -501.761,Z 1666.547,A 0.000,B 0.000,C 90.000,E1 98.454} C_DIS
LIN {X 0.149,Y -503.685,Z 1666.546,A 0.000,B 0.000,C 90.000,E1 98.219} C_DIS
LIN {X 0.011,Y -505.391,Z 1666.544,A 0.000,B 0.000,C 90.000,E1 97.992} C_DIS
LIN {X -0.056,Y -506.665,Z 1666.543,A 0.000,B 0.000,C 90.000,E1 97.757} C_DIS
LIN {X -0.241,Y -508.220,Z 1666.540,A 0.000,B 0.000,C 90.000,E1 97.296} C_DIS
LIN {X 0.086,Y -508.688,Z 1666.538,A 0.000,B 0.000,C 90.000,E1 96.777} C_DIS
LIN {X -0.083,Y -508.147,Z 1666.535,A 0.000,B 0.000,C 90.000,E1 96.315} C_DIS
LIN {X 0.254,Y -506.505,Z 1666.532,A 0.000,B 0.000,C 90.000,E1 95.796} C_DIS
LIN {X 0.144,Y -505.178,Z 1666.531,A 0.000,B 0.000,C 90.000,E1 95.568} C_DIS
LIN {X -0.081,Y -493.005,Z 1666.522,A 0.000,B 0.000,C 90.000,E1 93.898} C_DIS
LIN {X 0.045,Y -482.458,Z 1666.513,A 0.000,B 0.000,C 90.000,E1 92.407} C_DIS
LIN {X -0.007,Y -471.675,Z 1666.505,A 0.000,B 0.000,C 90.000,E1 90.917} C_DIS
LIN {X -0.212,Y -457.233,Z 1666.494,A 0.000,B 0.000,C 90.000,E1 88.912} C_DIS
LIN {X 0.219,Y -446.159,Z 1666.485,A 0.000,B 0.000,C 90.000,E1 87.306} C_DIS
LIN {X 0.033,Y -434.598,Z 1666.476,A 0.000,B 0.000,C 90.000,E1 85.755} C_DIS
LIN {X -0.185,Y -421.147,Z 1666.466,A 0.000,B 0.000,C 90.000,E1 83.913} C_DIS
LIN {X 0.063,Y -402.411,Z 1666.451,A 0.000,B 0.000,C 90.000,E1 81.141} C_DIS
LIN {X -0.096,Y -386.584,Z 1666.437,A 0.000,B 0.000,C 90.000,E1 78.634} C_DIS
LIN {X -0.133,Y -371.383,Z 1666.422,A 0.000,B 0.000,C 90.000,E1 76.047} C_DIS
LIN {X -0.037,Y -356.705,Z 1666.408,A 0.000,B 0.000,C 90.000,E1 73.378} C_DIS
LIN {X -0.127,Y -339.770,Z 1666.389,A 0.000,B 0.000,C 90.000,E1 70.061} C_DIS
LIN {X 0.109,Y -328.250,Z 1666.375,A 0.000,B 0.000,C 90.000,E1 67.539} C_DIS
LIN {X -0.048,Y -315.805,Z 1666.359,A 0.000,B 0.000,C 90.000,E1 64.717} C_DIS
LIN {X 0.102,Y -304.983,Z 1666.345,A 0.000,B 0.000,C 90.000,E1 62.103} C_DIS
LIN {X 0.116,Y -296.859,Z 1666.334,A 0.000,B 0.000,C 90.000,E1 60.127} C_DIS
LIN {X 0.130,Y -288.487,Z 1666.323,A 0.000,B 0.000,C 90.000,E1 58.122} C_DIS
LIN {X 0.136,Y -279.836,Z 1666.312,A 0.000,B 0.000,C 90.000,E1 56.087} C_DIS
LIN {X -0.008,Y -269.665,Z 1666.298,A 0.000,B 0.000,C 90.000,E1 53.703} C_DIS
LIN {X 0.057,Y -257.022,Z 1666.281,A 0.000,B 0.000,C 90.000,E1 50.517} C_DIS
LIN {X -0.130,Y -245.183,Z 1666.263,A 0.000,B 0.000,C 90.000,E1 47.310} C_DIS
LIN {X 0.035,Y -234.419,Z 1666.244,A 0.000,B 0.000,C 90.000,E1 43.947} C_DIS
LIN {X -0.018,Y -225.515,Z 1666.227,A 0.000,B 0.000,C 90.000,E1 40.943} C_DIS
LIN {X -0.061,Y -217.329,Z 1666.210,A 0.000,B 0.000,C 90.000,E1 37.890} C_DIS
LIN {X 0.065,Y -209.769,Z 1666.193,A 0.000,B 0.000,C 90.000,E1 34.739} C_DIS
LIN {X -0.015,Y -202.801,Z 1666.176,A 0.000,B 0.000,C 90.000,E1 31.592} C_DIS
LIN {X 0.046,Y -196.366,Z 1666.158,A 0.000,B 0.000,C 90.000,E1 28.359} C_DIS
LIN {X 0.025,Y -190.505,Z 1666.140,A 0.000,B 0.000,C 90.000,E1 25.103} C_DIS
LIN {X 0.052,Y -185.342,Z 1666.121,A 0.000,B 0.000,C 90.000,E1 21.791} C_DIS
LIN {X -0.020,Y -180.797,Z 1666.103,A 0.000,B 0.000,C 90.000,E1 18.471} C_DIS
LIN {X 0.074,Y -176.934,Z 1666.084,A 0.000,B 0.000,C 90.000,E1 15.064} C_DIS
LIN {X -0.034,Y -173.107,Z 1666.060,A 0.000,B 0.000,C 90.000,E1 10.838} C_DIS
LIN {X -0.048,Y -169.782,Z 1666.031,A 0.000,B 0.000,C 90.000,E1 5.682} C_DIS
LIN {X -0.031,Y -167.543,Z 1665.997,A 0.000,B 0.000,C 90.000,E1 359.542} C_DIS
LIN {X -0.012,Y -168.377,Z 1665.930,A 0.000,B 0.000,C 90.000,E1 347.353} C_DIS
LIN {X 0.066,Y -171.144,Z 1665.901,A 0.000,B 0.000,C 90.000,E1 342.127} C_DIS
LIN {X -0.011,Y -174.740,Z 1665.877,A 0.000,B 0.000,C 90.000,E1 337.847} C_DIS
LIN {X 0.059,Y -178.599,Z 1665.858,A 0.000,B 0.000,C 90.000,E1 334.409} C_DIS
LIN {X -0.029,Y -183.189,Z 1665.839,A 0.000,B 0.000,C 90.000,E1 331.051} C_DIS
LIN {X -0.053,Y -188.616,Z 1665.821,A 0.000,B 0.000,C 90.000,E1 327.709} C_DIS
LIN {X 0.090,Y -193.396,Z 1665.807,A 0.000,B 0.000,C 90.000,E1 325.182} C_DIS
LIN {X -0.046,Y -198.727,Z 1665.793,A 0.000,B 0.000,C 90.000,E1 322.763} C_DIS
LIN {X 0.050,Y -205.808,Z 1665.777,A 0.000,B 0.000,C 90.000,E1 319.908} C_DIS
LIN {X 0.020,Y -214.971,Z 1665.760,A 0.000,B 0.000,C 90.000,E1 316.743} C_DIS
LIN {X -0.019,Y -224.107,Z 1665.745,A 0.000,B 0.000,C 90.000,E1 314.028} C_DIS
LIN {X -0.005,Y -234.235,Z 1665.730,A 0.000,B 0.000,C 90.000,E1 311.353} C_DIS
LIN {X -0.059,Y -245.532,Z 1665.715,A 0.000,B 0.000,C 90.000,E1 308.749} C_DIS
LIN {X 0.020,Y -256.531,Z 1665.703,A 0.000,B 0.000,C 90.000,E1 306.537} C_DIS
LIN {X -0.068,Y -272.859,Z 1665.687,A 0.000,B 0.000,C 90.000,E1 303.706} C_DIS
LIN {X 0.036,Y -291.003,Z 1665.672,A 0.000,B 0.000,C 90.000,E1 300.924} C_DIS
LIN {X -0.094,Y -310.441,Z 1665.657,A 0.000,B 0.000,C 90.000,E1 298.281} C_DIS
LIN {X 0.159,Y -323.054,Z 1665.648,A 0.000,B 0.000,C 90.000,E1 296.616} C_DIS
LIN {X -0.119,Y -335.361,Z 1665.639,A 0.000,B 0.000,C 90.000,E1 295.079} C_DIS
LIN {X -0.034,Y -350.168,Z 1665.629,A 0.000,B 0.000,C 90.000,E1 293.206} C_DIS
LIN {X -0.183,Y -362.425,Z 1665.620,A 0.000,B 0.000,C 90.000,E1 291.716} C_DIS
LIN {X 0.101,Y -371.968,Z 1665.614,A 0.000,B 0.000,C 90.000,E1 290.482} C_DIS
LIN {X -0.090,Y -378.745,Z 1665.609,A 0.000,B 0.000,C 90.000,E1 289.631} C_DIS
LIN {X 0.149,Y -384.975,Z 1665.604,A 0.000,B 0.000,C 90.000,E1 288.725} C_DIS
LIN {X -0.067,Y -388.821,Z 1665.601,A 0.000,B 0.000,C 90.000,E1 288.181} C_DIS
LIN {X -0.109,Y -393.835,Z 1665.596,A 0.000,B 0.000,C 90.000,E1 287.330} C_DIS
LIN {X 0.162,Y -397.968,Z 1665.591,A 0.000,B 0.000,C 90.000,E1 286.441} C_DIS
LIN {X 0.092,Y -401.283,Z 1665.587,A 0.000,B 0.000,C 90.000,E1 285.607} C_DIS
LIN {X -0.032,Y -403.036,Z 1665.584,A 0.000,B 0.000,C 90.000,E1 285.064} C_DIS
LIN {X 0.135,Y -404.419,Z 1665.581,A 0.000,B 0.000,C 90.000,E1 284.481} C_DIS
LIN {X 0.023,Y -405.388,Z 1665.578,A 0.000,B 0.000,C 90.000,E1 283.939} C_DIS
LIN {X -0.180,Y -405.946,Z 1665.574,A 0.000,B 0.000,C 90.000,E1 283.411} C_DIS
LIN {X 0.017,Y -406.083,Z 1665.571,A 0.000,B 0.000,C 90.000,E1 282.827} C_DIS
LIN {X -0.175,Y -405.716,Z 1665.568,A 0.000,B 0.000,C 90.000,E1 282.299} C_DIS
LIN {X 0.030,Y -404.929,Z 1665.565,A 0.000,B 0.000,C 90.000,E1 281.715} C_DIS
LIN {X -0.164,Y -403.567,Z 1665.562,A 0.000,B 0.000,C 90.000,E1 281.186} C_DIS
LIN {X 0.032,Y -401.680,Z 1665.559,A 0.000,B 0.000,C 90.000,E1 280.602} C_DIS
LIN {X 0.218,Y -399.190,Z 1665.556,A 0.000,B 0.000,C 90.000,E1 280.018} C_DIS
LIN {X -0.002,Y -394.385,Z 1665.551,A 0.000,B 0.000,C 90.000,E1 279.208} C_DIS
LIN {X 0.137,Y -388.645,Z 1665.547,A 0.000,B 0.000,C 90.000,E1 278.341} C_DIS
LIN {X -0.160,Y -382.157,Z 1665.542,A 0.000,B 0.000,C 90.000,E1 277.530} C_DIS
LIN {X -0.102,Y -377.296,Z 1665.538,A 0.000,B 0.000,C 90.000,E1 276.947} C_DIS
LIN {X -0.052,Y -371.909,Z 1665.535,A 0.000,B 0.000,C 90.000,E1 276.372} C_DIS
LIN {X 0.167,Y -366.100,Z 1665.532,A 0.000,B 0.000,C 90.000,E1 275.796} C_DIS
LIN {X -0.101,Y -359.957,Z 1665.530,A 0.000,B 0.000,C 90.000,E1 275.334} C_DIS
LIN {X -0.095,Y -353.504,Z 1665.527,A 0.000,B 0.000,C 90.000,E1 274.878} C_DIS
LIN {X -0.083,Y -347.004,Z 1665.525,A 0.000,B 0.000,C 90.000,E1 274.473} C_DIS
LIN {X 0.140,Y -337.300,Z 1665.522,A 0.000,B 0.000,C 90.000,E1 273.898} C_DIS
LIN {X -0.014,Y -327.702,Z 1665.519,A 0.000,B 0.000,C 90.000,E1 273.440} C_DIS
LIN {X 0.066,Y -317.776,Z 1665.517,A 0.000,B 0.000,C 90.000,E1 272.980} C_DIS
LIN {X 0.075,Y -307.647,Z 1665.514,A 0.000,B 0.000,C 90.000,E1 272.579} C_DIS
LIN {X 0.069,Y -297.065,Z 1665.512,A 0.000,B 0.000,C 90.000,E1 272.236} C_DIS
LIN {X -0.122,Y -285.836,Z 1665.511,A 0.000,B 0.000,C 90.000,E1 272.007} C_DIS
LIN {X 0.042,Y -277.501,Z 1665.510,A 0.000,B 0.000,C 90.000,E1 271.835} C_DIS
LIN {X 0.053,Y -266.547,Z 1665.510,A 0.000,B 0.000,C 90.000,E1 271.718} C_DIS
LIN {X 0.085,Y -233.275,Z 1665.509,A 0.000,B 0.000,C 90.000,E1 271.547} C_DIS
LIN {X -0.088,Y -182.933,Z 1665.507,A 0.000,B 0.000,C 90.000,E1 271.375} C_DIS
LIN {X 0.075,Y -181.383,Z 1665.507,A 0.000,B 0.000,C 90.000,E1 271.318} C_DIS
LIN {X -0.053,Y -181.580,Z 1665.502,A 0.000,B 0.000,C 90.000,E1 270.344} C_DIS
LIN {X -0.048,Y -180.883,Z 1665.473,A 0.000,B 0.000,C 90.000,E1 265.122} C_DIS
LIN {X 0.011,Y -179.003,Z 1665.445,A 0.000,B 0.000,C 90.000,E1 260.038} C_DIS
LIN {X -0.071,Y -178.603,Z 1665.440,A 0.000,B 0.000,C 90.000,E1 259.218} C_DIS
LIN {X -0.002,Y -175.655,Z 1665.412,A 0.000,B 0.000,C 90.000,E1 254.102} C_DIS
LIN {X 0.004,Y -172.374,Z 1665.388,A 0.000,B 0.000,C 90.000,E1 249.826} C_DIS
LIN {X 0.018,Y -171.168,Z 1665.378,A 0.000,B 0.000,C 90.000,E1 248.103} C_DIS
LIN {X 0.062,Y -167.465,Z 1665.354,A 0.000,B 0.000,C 90.000,E1 243.768} C_DIS
LIN {X -0.005,Y -166.862,Z 1665.350,A 0.000,B 0.000,C 90.000,E1 242.922} C_DIS
LIN {X 0.049,Y -162.165,Z 1665.320,A 0.000,B 0.000,C 90.000,E1 237.661} C_DIS
LIN {X -0.031,Y -160.727,Z 1665.311,A 0.000,B 0.000,C 90.000,E1 235.928} C_DIS
LIN {X -0.050,Y -157.530,Z 1665.291,A 0.000,B 0.000,C 90.000,E1 232.396} C_DIS
LIN {X 0.007,Y -155.557,Z 1665.276,A 0.000,B 0.000,C 90.000,E1 229.703} C_DIS
LIN {X -0.059,Y -151.847,Z 1665.251,A 0.000,B 0.000,C 90.000,E1 225.243} C_DIS
LIN {X -0.045,Y -150.066,Z 1665.236,A 0.000,B 0.000,C 90.000,E1 222.528} C_DIS
LIN {X -0.011,Y -146.875,Z 1665.211,A 0.000,B 0.000,C 90.000,E1 217.971} C_DIS
LIN {X -0.022,Y -145.459,Z 1665.196,A 0.000,B 0.000,C 90.000,E1 215.231} C_DIS
LIN {X 0.019,Y -142.875,Z 1665.170,A 0.000,B 0.000,C 90.000,E1 210.620} C_DIS
LIN {X 0.017,Y -141.493,Z 1665.150,A 0.000,B 0.000,C 90.000,E1 206.924} C_DIS
LIN {X 0.003,Y -139.386,Z 1665.114,A 0.000,B 0.000,C 90.000,E1 200.429} C_DIS
LIN {X -0.009,Y -138.842,Z 1665.098,A 0.000,B 0.000,C 90.000,E1 197.638} C_DIS
LIN {X 0.051,Y -138.353,Z 1665.056,A 0.000,B 0.000,C 90.000,E1 190.141} C_DIS
LIN {X 0.047,Y -139.519,Z 1665.005,A 0.000,B 0.000,C 90.000,E1 180.802} C_DIS
LIN {X -0.012,Y -141.180,Z 1664.974,A 0.000,B 0.000,C 90.000,E1 175.241} C_DIS
LIN {X -0.041,Y -142.558,Z 1664.958,A 0.000,B 0.000,C 90.000,E1 172.470} C_DIS
LIN {X 0.025,Y -144.839,Z 1664.932,A 0.000,B 0.000,C 90.000,E1 167.825} C_DIS
LIN {X 0.011,Y -147.463,Z 1664.912,A 0.000,B 0.000,C 90.000,E1 164.157} C_DIS
LIN {X 0.038,Y -150.046,Z 1664.892,A 0.000,B 0.000,C 90.000,E1 160.496} C_DIS
LIN {X 0.043,Y -153.388,Z 1664.872,A 0.000,B 0.000,C 90.000,E1 156.869} C_DIS
LIN {X -0.050,Y -155.919,Z 1664.857,A 0.000,B 0.000,C 90.000,E1 154.204} C_DIS
LIN {X 0.064,Y -159.784,Z 1664.837,A 0.000,B 0.000,C 90.000,E1 150.589} C_DIS
LIN {X -0.088,Y -162.025,Z 1664.827,A 0.000,B 0.000,C 90.000,E1 148.869} C_DIS
LIN {X 0.025,Y -166.219,Z 1664.807,A 0.000,B 0.000,C 90.000,E1 145.308} C_DIS
LIN {X 0.027,Y -171.236,Z 1664.788,A 0.000,B 0.000,C 90.000,E1 141.823} C_DIS
LIN {X -0.050,Y -176.122,Z 1664.769,A 0.000,B 0.000,C 90.000,E1 138.405} C_DIS
LIN {X 0.067,Y -180.388,Z 1664.755,A 0.000,B 0.000,C 90.000,E1 135.810} C_DIS
LIN {X 0.043,Y -185.796,Z 1664.736,A 0.000,B 0.000,C 90.000,E1 132.447} C_DIS
LIN {X -0.024,Y -190.413,Z 1664.722,A 0.000,B 0.000,C 90.000,E1 129.967} C_DIS
LIN {X -0.009,Y -197.737,Z 1664.699,A 0.000,B 0.000,C 90.000,E1 125.851} C_DIS
LIN {X 0.081,Y -200.983,Z 1664.690,A 0.000,B 0.000,C 90.000,E1 124.199} C_DIS
LIN {X 0.097,Y -207.258,Z 1664.671,A 0.000,B 0.000,C 90.000,E1 120.797} C_DIS
LIN {X 0.076,Y -207.528,Z 1664.671,A 0.000,B 0.000,C 90.000,E1 120.669} C_DIS
LIN {X 0.086,Y -328.653,Z 1664.670,A 0.000,B 0.000,C 90.000,E1 120.669} C_DIS
LIN {X -0.060,Y -330.515,Z 1664.670,A 0.000,B 0.000,C 90.000,E1 120.669} C_DIS
LIN {X -0.180,Y -335.594,Z 1664.669,A 0.000,B 0.000,C 90.000,E1 120.463} C_DIS
LIN {X -0.009,Y -338.296,Z 1664.668,A 0.000,B 0.000,C 90.000,E1 120.207} C_DIS
LIN {X -0.124,Y -342.049,Z 1664.665,A 0.000,B 0.000,C 90.000,E1 119.745} C_DIS
LIN {X 0.023,Y -343.730,Z 1664.663,A 0.000,B 0.000,C 90.000,E1 119.411} C_DIS
LIN {X 0.045,Y -357.579,Z 1664.646,A 0.000,B 0.000,C 90.000,E1 116.360} C_DIS
LIN {X -0.058,Y -371.571,Z 1664.632,A 0.000,B 0.000,C 90.000,E1 113.695} C_DIS
LIN {X 0.000,Y -385.356,Z 1664.619,A 0.000,B 0.000,C 90.000,E1 111.354} C_DIS
LIN {X -0.092,Y -400.510,Z 1664.606,A 0.000,B 0.000,C 90.000,E1 109.087} C_DIS
LIN {X -0.080,Y -417.137,Z 1664.594,A 0.000,B 0.000,C 90.000,E1 106.858} C_DIS
LIN {X 0.113,Y -435.352,Z 1664.582,A 0.000,B 0.000,C 90.000,E1 104.662} C_DIS
LIN {X -0.001,Y -455.018,Z 1664.570,A 0.000,B 0.000,C 90.000,E1 102.591} C_DIS
LIN {X 0.082,Y -475.320,Z 1664.559,A 0.000,B 0.000,C 90.000,E1 100.658} C_DIS
LIN {X 0.223,Y -501.315,Z 1664.547,A 0.000,B 0.000,C 90.000,E1 98.454} C_DIS
LIN {X 0.044,Y -504.896,Z 1664.545,A 0.000,B 0.000,C 90.000,E1 98.049} C_DIS
LIN {X -0.025,Y -506.247,Z 1664.543,A 0.000,B 0.000,C 90.000,E1 97.814} C_DIS
LIN {X -0.162,Y -507.237,Z 1664.542,A 0.000,B 0.000,C 90.000,E1 97.587} C_DIS
LIN {X 0.164,Y -508.329,Z 1664.539,A 0.000,B 0.000,C 90.000,E1 97.068} C_DIS
LIN {X -0.009,Y -508.390,Z 1664.537,A 0.000,B 0.000,C 90.000,E1 96.606} C_DIS
LIN {X -0.177,Y -507.426,Z 1664.534,A 0.000,B 0.000,C 90.000,E1 96.144} C_DIS
LIN {X -0.234,Y -506.516,Z 1664.533,A 0.000,B 0.000,C 90.000,E1 95.910} C_DIS
LIN {X 0.160,Y -505.264,Z 1664.531,A 0.000,B 0.000,C 90.000,E1 95.625} C_DIS
LIN {X 0.029,Y -494.885,Z 1664.523,A 0.000,B 0.000,C 90.000,E1 94.188} C_DIS
LIN {X 0.216,Y -484.412,Z 1664.515,A 0.000,B 0.000,C 90.000,E1 92.694} C_DIS
LIN {X 0.192,Y -473.698,Z 1664.507,A 0.000,B 0.000,C 90.000,E1 91.203} C_DIS
LIN {X 0.024,Y -459.249,Z 1664.496,A 0.000,B 0.000,C 90.000,E1 89.198} C_DIS
LIN {X 0.041,Y -448.218,Z 1664.487,A 0.000,B 0.000,C 90.000,E1 87.650} C_DIS
LIN {X -0.134,Y -436.734,Z 1664.478,A 0.000,B 0.000,C 90.000,E1 86.102} C_DIS
LIN {X 0.109,Y -423.245,Z 1664.468,A 0.000,B 0.000,C 90.000,E1 84.204} C_DIS
LIN {X 0.000,Y -404.355,Z 1664.453,A 0.000,B 0.000,C 90.000,E1 81.489} C_DIS
LIN {X -0.132,Y -386.679,Z 1664.437,A 0.000,B 0.000,C 90.000,E1 78.701} C_DIS
LIN {X -0.173,Y -371.465,Z 1664.423,A 0.000,B 0.000,C 90.000,E1 76.117} C_DIS
LIN {X -0.043,Y -358.373,Z 1664.410,A 0.000,B 0.000,C 90.000,E1 73.740} C_DIS
LIN {X -0.092,Y -342.803,Z 1664.393,A 0.000,B 0.000,C 90.000,E1 70.732} C_DIS
LIN {X 0.095,Y -331.147,Z 1664.379,A 0.000,B 0.000,C 90.000,E1 68.230} C_DIS
LIN {X -0.052,Y -317.211,Z 1664.362,A 0.000,B 0.000,C 90.000,E1 65.101} C_DIS
LIN {X 0.133,Y -306.333,Z 1664.347,A 0.000,B 0.000,C 90.000,E1 62.487} C_DIS
LIN {X 0.027,Y -298.244,Z 1664.336,A 0.000,B 0.000,C 90.000,E1 60.539} C_DIS
LIN {X 0.064,Y -289.913,Z 1664.325,A 0.000,B 0.000,C 90.000,E1 58.535} C_DIS
LIN {X 0.098,Y -281.329,Z 1664.314,A 0.000,B 0.000,C 90.000,E1 56.501} C_DIS
LIN {X -0.080,Y -269.684,Z 1664.299,A 0.000,B 0.000,C 90.000,E1 53.783} C_DIS
